// TIA Portal V20 export
FUNCTION "CollectAlarms" : Void   // FC62, LAD
TITLE = Alarm Collector Unit
// Collects alarms from the respective level and categorises the alarms into the different alarm classes.
// stored: Namespace Unit1, SetENOAutomatically false
   VAR_INPUT
      resetAlarms : Bool;
      disableAlarms : Bool;
   END_VAR
   VAR_OUTPUT
      commandsToUnit : "LUC_typeStateCommands";   // Feedback to the unit
   END_VAR
   VAR_TEMP
      interfaceUnuse : Array[0..1] of Bool;
      otherUnitError : Array[0..1] of Bool;
   END_VAR
   VAR CONSTANT
      TRUE : Bool := true;
      DelayTime : Time := T#300ms;
   END_VAR
BEGIN

REGION Network 1: Reset Alarms
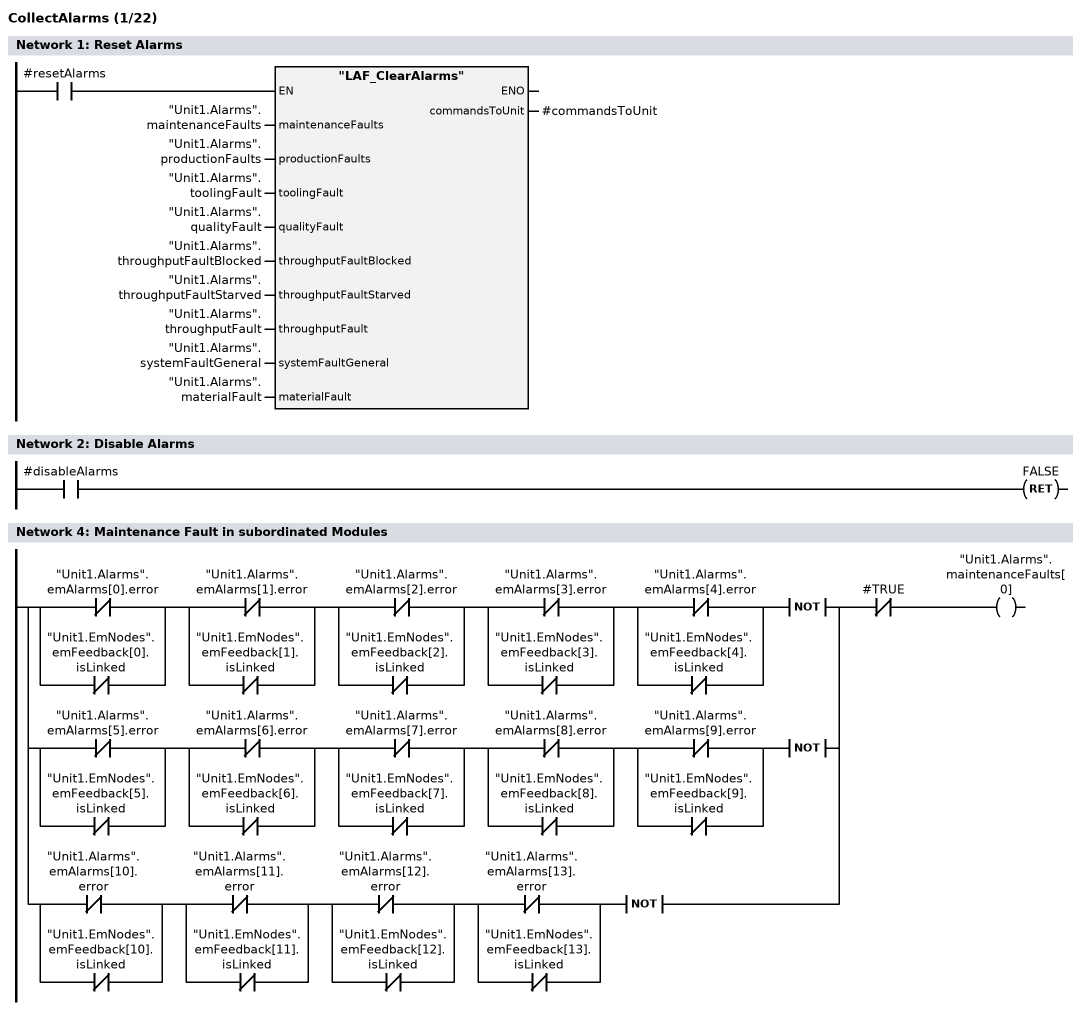
   RUNG wire#powerrail
      Contact( #resetAlarms )
      "LAF_ClearAlarms"(maintenanceFaults := "Unit1.Alarms".maintenanceFaults, productionFaults := "Unit1.Alarms".productionFaults, toolingFault := "Unit1.Alarms".toolingFault, qualityFault := "Unit1.Alarms".qualityFault, throughputFaultBlocked := "Unit1.Alarms".throughputFaultBlocked, throughputFaultStarved := "Unit1.Alarms".throughputFaultStarved, throughputFault := "Unit1.Alarms".throughputFault, systemFaultGeneral := "Unit1.Alarms".systemFaultGeneral, materialFault := "Unit1.Alarms".materialFault, commandsToUnit => #commandsToUnit)
   END_RUNG
   // the same network as SCL:
   IF #resetAlarms THEN
       "LAF_ClearAlarms"(maintenanceFaults := "Unit1.Alarms".maintenanceFaults,
                         productionFaults := "Unit1.Alarms".productionFaults,
                         toolingFault := "Unit1.Alarms".toolingFault,
                         qualityFault := "Unit1.Alarms".qualityFault,
                         throughputFaultBlocked := "Unit1.Alarms".throughputFaultBlocked,
                         throughputFaultStarved := "Unit1.Alarms".throughputFaultStarved,
                         throughputFault := "Unit1.Alarms".throughputFault,
                         systemFaultGeneral := "Unit1.Alarms".systemFaultGeneral,
                         materialFault := "Unit1.Alarms".materialFault,
                         commandsToUnit => #commandsToUnit);
   END_IF;
END_REGION

REGION Network 2: Disable Alarms
   RUNG wire#powerrail
      Contact( #disableAlarms )
      ReturnCoil( FALSE )
   END_RUNG
   // the same network as SCL:
   IF #disableAlarms THEN
       ENO := FALSE;
       RETURN;
   END_IF;
END_REGION

REGION Network 3: *************** Fault ************************
END_REGION

REGION Network 4: Maintenance Fault in subordinated Modules
   RUNG wire#powerrail
      I_Contact( "Unit1.Alarms".emAlarms[0].error )
      wire#w1
      I_Contact( "Unit1.Alarms".emAlarms[1].error )
      wire#w2
      I_Contact( "Unit1.Alarms".emAlarms[2].error )
      wire#w3
      I_Contact( "Unit1.Alarms".emAlarms[3].error )
      wire#w4
      I_Contact( "Unit1.Alarms".emAlarms[4].error )
      wire#w5
      Not()
      wire#w6
      I_Contact( #TRUE )
      Coil( "Unit1.Alarms".maintenanceFaults[0] )
   END_RUNG
   RUNG wire#powerrail
      I_Contact( "Unit1.EmNodes".emFeedback[0].isLinked )
   END_RUNG wire#w1
   RUNG wire#w1
      I_Contact( "Unit1.EmNodes".emFeedback[1].isLinked )
   END_RUNG wire#w2
   RUNG wire#w2
      I_Contact( "Unit1.EmNodes".emFeedback[2].isLinked )
   END_RUNG wire#w3
   RUNG wire#w3
      I_Contact( "Unit1.EmNodes".emFeedback[3].isLinked )
   END_RUNG wire#w4
   RUNG wire#w4
      I_Contact( "Unit1.EmNodes".emFeedback[4].isLinked )
   END_RUNG wire#w5
   RUNG wire#powerrail
      I_Contact( "Unit1.Alarms".emAlarms[5].error )
      wire#w7
      I_Contact( "Unit1.Alarms".emAlarms[6].error )
      wire#w8
      I_Contact( "Unit1.Alarms".emAlarms[7].error )
      wire#w9
      I_Contact( "Unit1.Alarms".emAlarms[8].error )
      wire#w10
      I_Contact( "Unit1.Alarms".emAlarms[9].error )
      wire#w11
      Not()
   END_RUNG wire#w6
   RUNG wire#powerrail
      I_Contact( "Unit1.EmNodes".emFeedback[5].isLinked )
   END_RUNG wire#w7
   RUNG wire#w7
      I_Contact( "Unit1.EmNodes".emFeedback[6].isLinked )
   END_RUNG wire#w8
   RUNG wire#w8
      I_Contact( "Unit1.EmNodes".emFeedback[7].isLinked )
   END_RUNG wire#w9
   RUNG wire#w9
      I_Contact( "Unit1.EmNodes".emFeedback[8].isLinked )
   END_RUNG wire#w10
   RUNG wire#w10
      I_Contact( "Unit1.EmNodes".emFeedback[9].isLinked )
   END_RUNG wire#w11
   RUNG wire#powerrail
      I_Contact( "Unit1.Alarms".emAlarms[10].error )
      wire#w12
      I_Contact( "Unit1.Alarms".emAlarms[11].error )
      wire#w13
      I_Contact( "Unit1.Alarms".emAlarms[12].error )
      wire#w14
      I_Contact( "Unit1.Alarms".emAlarms[13].error )
      wire#w15
      Not()
   END_RUNG wire#w6
   RUNG wire#powerrail
      I_Contact( "Unit1.EmNodes".emFeedback[10].isLinked )
   END_RUNG wire#w12
   RUNG wire#w12
      I_Contact( "Unit1.EmNodes".emFeedback[11].isLinked )
   END_RUNG wire#w13
   RUNG wire#w13
      I_Contact( "Unit1.EmNodes".emFeedback[12].isLinked )
   END_RUNG wire#w14
   RUNG wire#w14
      I_Contact( "Unit1.EmNodes".emFeedback[13].isLinked )
   END_RUNG wire#w15
   // the same network as SCL:
   "Unit1.Alarms".maintenanceFaults[0] := (NOT ((NOT "Unit1.Alarms".emAlarms[0].error OR NOT "Unit1.EmNodes".emFeedback[0].isLinked) AND (NOT "Unit1.Alarms".emAlarms[1].error OR NOT "Unit1.EmNodes".emFeedback[1].isLinked) AND (NOT "Unit1.Alarms".emAlarms[2].error OR NOT "Unit1.EmNodes".emFeedback[2].isLinked) AND (NOT "Unit1.Alarms".emAlarms[3].error OR NOT "Unit1.EmNodes".emFeedback[3].isLinked) AND (NOT "Unit1.Alarms".emAlarms[4].error OR NOT "Unit1.EmNodes".emFeedback[4].isLinked)) OR NOT ((NOT "Unit1.Alarms".emAlarms[5].error OR NOT "Unit1.EmNodes".emFeedback[5].isLinked) AND (NOT "Unit1.Alarms".emAlarms[6].error OR NOT "Unit1.EmNodes".emFeedback[6].isLinked) AND (NOT "Unit1.Alarms".emAlarms[7].error OR NOT "Unit1.EmNodes".emFeedback[7].isLinked) AND (NOT "Unit1.Alarms".emAlarms[8].error OR NOT "Unit1.EmNodes".emFeedback[8].isLinked) AND (NOT "Unit1.Alarms".emAlarms[9].error OR NOT "Unit1.EmNodes".emFeedback[9].isLinked)) OR NOT ((NOT "Unit1.Alarms".emAlarms[10].error OR NOT "Unit1.EmNodes".emFeedback[10].isLinked) AND (NOT "Unit1.Alarms".emAlarms[11].error OR NOT "Unit1.EmNodes".emFeedback[11].isLinked) AND (NOT "Unit1.Alarms".emAlarms[12].error OR NOT "Unit1.EmNodes".emFeedback[12].isLinked) AND (NOT "Unit1.Alarms".emAlarms[13].error OR NOT "Unit1.EmNodes".emFeedback[13].isLinked))) AND NOT #TRUE;
END_REGION

REGION Network 5: PFE Maintenance Faults 0 ~ 29
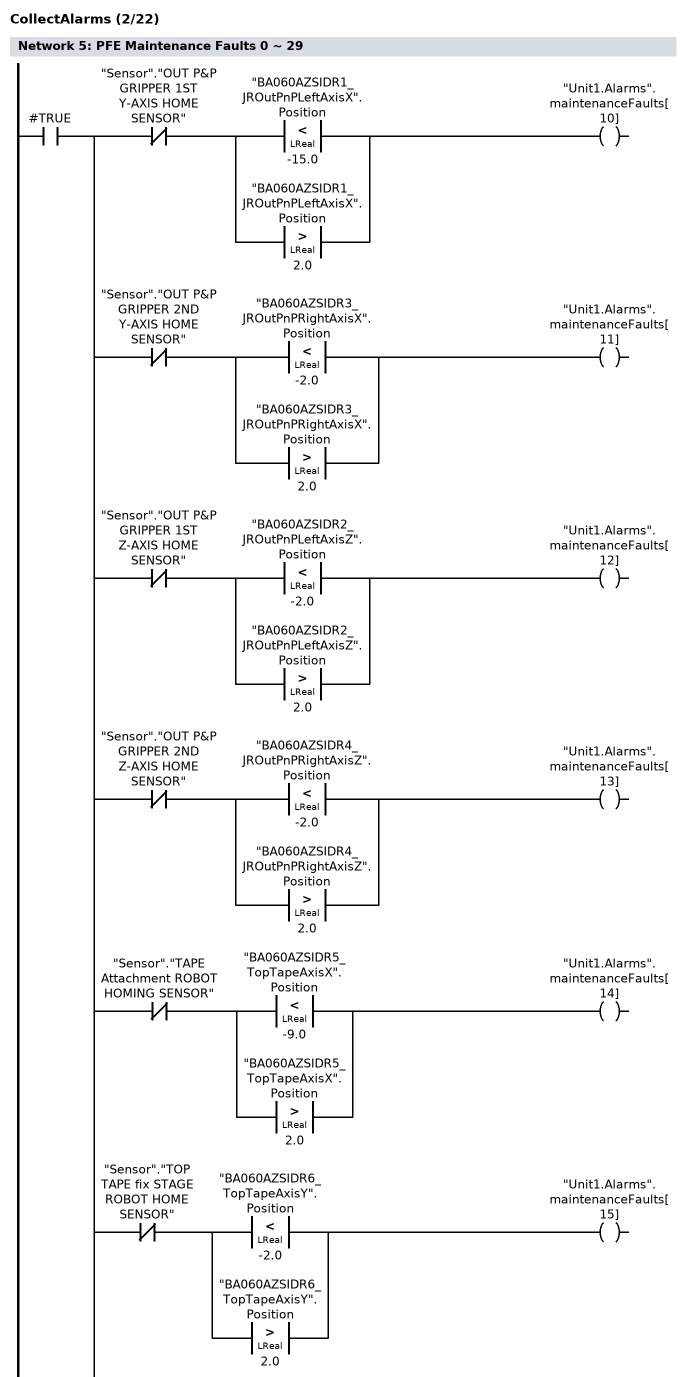
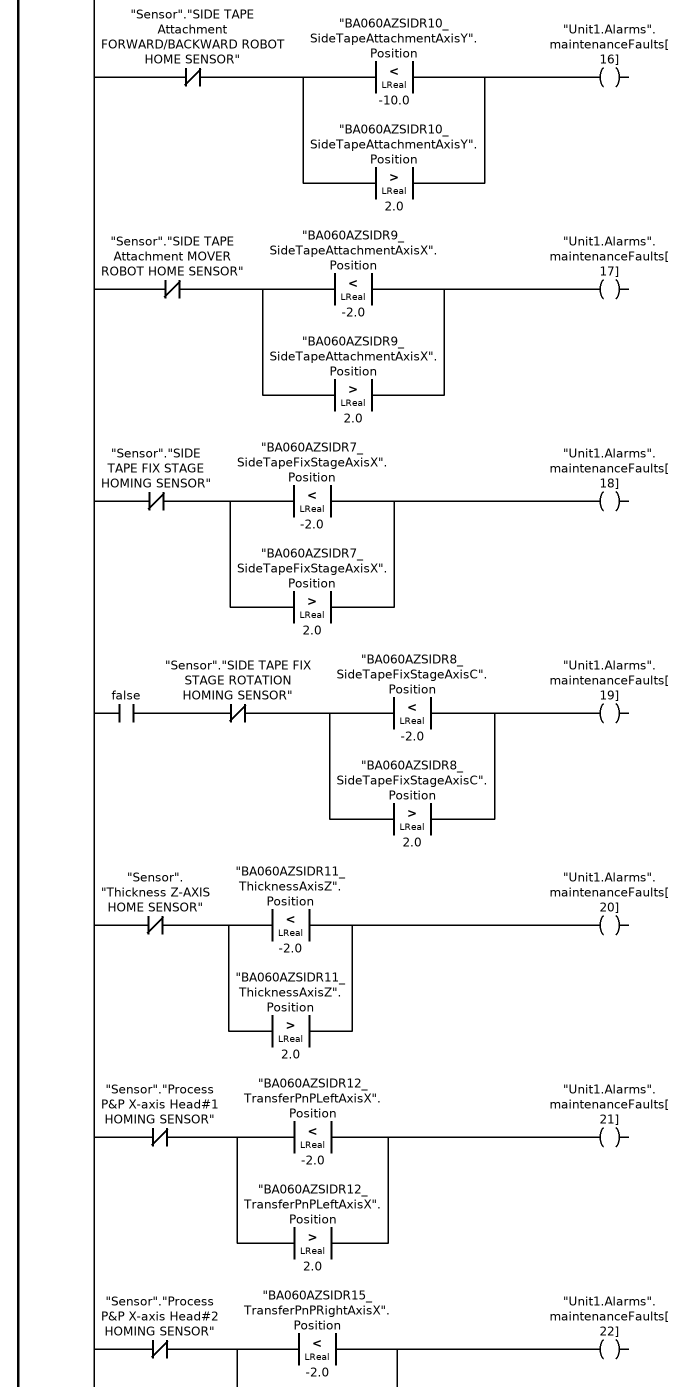
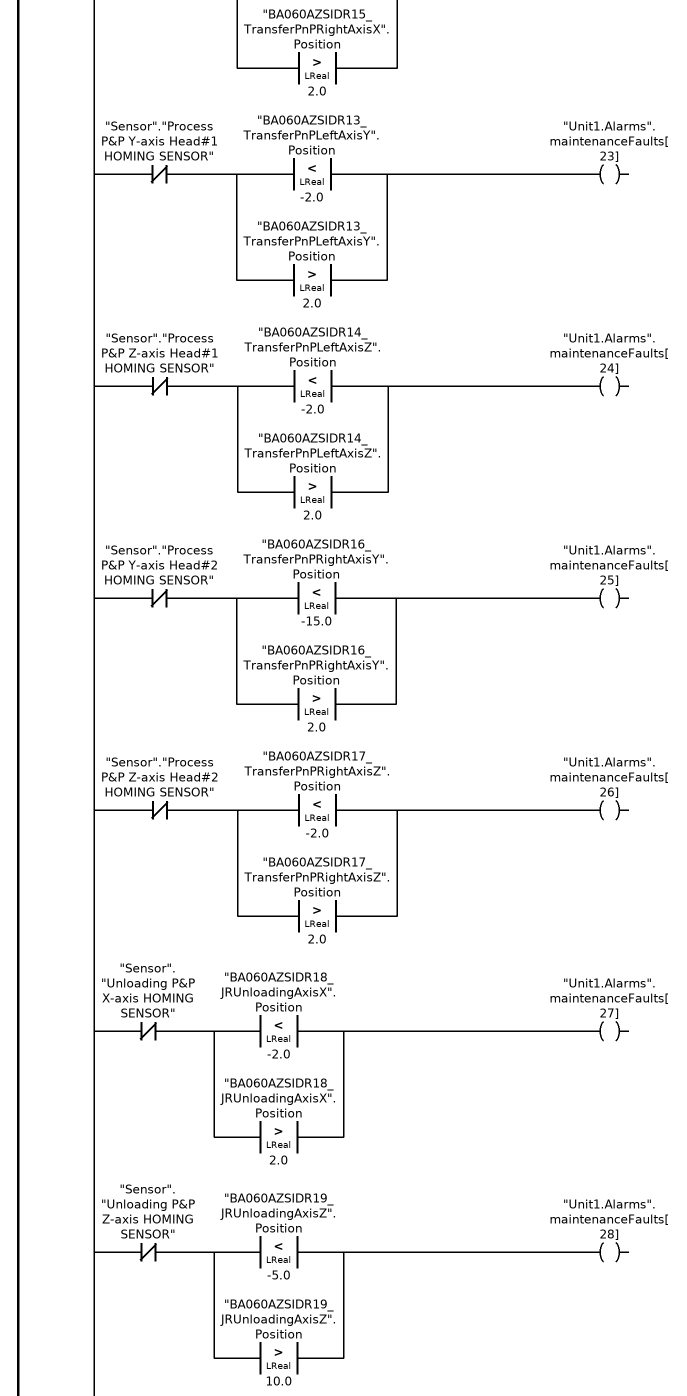
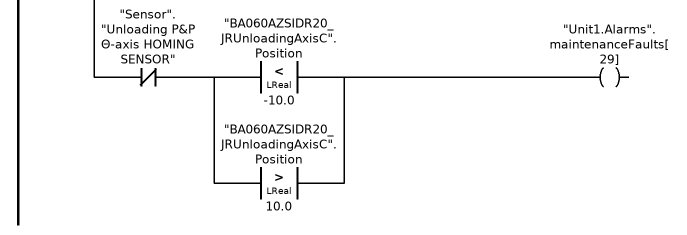
   RUNG wire#powerrail
      Contact( #TRUE )
      wire#w1
      I_Contact( "Sensor"."OUT P&P GRIPPER 1ST Y-AXIS HOME SENSOR" )
      wire#w2
      { S7_Templates := "SrcType := LReal" } LT_Contact(in1 := "BA060AZSIDR1_JROutPnPLeftAxisX".Position, in2 := -15.0)
      wire#w3
      Coil( "Unit1.Alarms".maintenanceFaults[10] )
   END_RUNG
   RUNG wire#w2
      { S7_Templates := "SrcType := LReal" } GT_Contact(in1 := "BA060AZSIDR1_JROutPnPLeftAxisX".Position, in2 := 2.0)
   END_RUNG wire#w3
   RUNG wire#w1
      I_Contact( "Sensor"."OUT P&P GRIPPER 2ND Y-AXIS HOME SENSOR" )
      wire#w4
      { S7_Templates := "SrcType := LReal" } LT_Contact(in1 := "BA060AZSIDR3_JROutPnPRightAxisX".Position, in2 := -2.0)
      wire#w5
      Coil( "Unit1.Alarms".maintenanceFaults[11] )
   END_RUNG
   RUNG wire#w4
      { S7_Templates := "SrcType := LReal" } GT_Contact(in1 := "BA060AZSIDR3_JROutPnPRightAxisX".Position, in2 := 2.0)
   END_RUNG wire#w5
   RUNG wire#w1
      I_Contact( "Sensor"."OUT P&P GRIPPER 1ST Z-AXIS HOME SENSOR" )
      wire#w6
      { S7_Templates := "SrcType := LReal" } LT_Contact(in1 := "BA060AZSIDR2_JROutPnPLeftAxisZ".Position, in2 := -2.0)
      wire#w7
      Coil( "Unit1.Alarms".maintenanceFaults[12] )
   END_RUNG
   RUNG wire#w6
      { S7_Templates := "SrcType := LReal" } GT_Contact(in1 := "BA060AZSIDR2_JROutPnPLeftAxisZ".Position, in2 := 2.0)
   END_RUNG wire#w7
   RUNG wire#w1
      I_Contact( "Sensor"."OUT P&P GRIPPER 2ND Z-AXIS HOME SENSOR" )
      wire#w8
      { S7_Templates := "SrcType := LReal" } LT_Contact(in1 := "BA060AZSIDR4_JROutPnPRightAxisZ".Position, in2 := -2.0)
      wire#w9
      Coil( "Unit1.Alarms".maintenanceFaults[13] )
   END_RUNG
   RUNG wire#w8
      { S7_Templates := "SrcType := LReal" } GT_Contact(in1 := "BA060AZSIDR4_JROutPnPRightAxisZ".Position, in2 := 2.0)
   END_RUNG wire#w9
   RUNG wire#w1
      I_Contact( "Sensor"."TAPE  Attachment ROBOT HOMING SENSOR" )
      wire#w10
      { S7_Templates := "SrcType := LReal" } LT_Contact(in1 := "BA060AZSIDR5_TopTapeAxisX".Position, in2 := -9.0)
      wire#w11
      Coil( "Unit1.Alarms".maintenanceFaults[14] )
   END_RUNG
   RUNG wire#w10
      { S7_Templates := "SrcType := LReal" } GT_Contact(in1 := "BA060AZSIDR5_TopTapeAxisX".Position, in2 := 2.0)
   END_RUNG wire#w11
   RUNG wire#w1
      I_Contact( "Sensor"."TOP TAPE fix STAGE ROBOT HOME SENSOR" )
      wire#w12
      { S7_Templates := "SrcType := LReal" } LT_Contact(in1 := "BA060AZSIDR6_TopTapeAxisY".Position, in2 := -2.0)
      wire#w13
      Coil( "Unit1.Alarms".maintenanceFaults[15] )
   END_RUNG
   RUNG wire#w12
      { S7_Templates := "SrcType := LReal" } GT_Contact(in1 := "BA060AZSIDR6_TopTapeAxisY".Position, in2 := 2.0)
   END_RUNG wire#w13
   RUNG wire#w1
      I_Contact( "Sensor"."SIDE TAPE Attachment FORWARD/BACKWARD ROBOT HOME SENSOR" )
      wire#w14
      { S7_Templates := "SrcType := LReal" } LT_Contact(in1 := "BA060AZSIDR10_SideTapeAttachmentAxisY".Position, in2 := -10.0)
      wire#w15
      Coil( "Unit1.Alarms".maintenanceFaults[16] )
   END_RUNG
   RUNG wire#w14
      { S7_Templates := "SrcType := LReal" } GT_Contact(in1 := "BA060AZSIDR10_SideTapeAttachmentAxisY".Position, in2 := 2.0)
   END_RUNG wire#w15
   RUNG wire#w1
      I_Contact( "Sensor"."SIDE TAPE Attachment MOVER ROBOT HOME SENSOR" )
      wire#w16
      { S7_Templates := "SrcType := LReal" } LT_Contact(in1 := "BA060AZSIDR9_SideTapeAttachmentAxisX".Position, in2 := -2.0)
      wire#w17
      Coil( "Unit1.Alarms".maintenanceFaults[17] )
   END_RUNG
   RUNG wire#w16
      { S7_Templates := "SrcType := LReal" } GT_Contact(in1 := "BA060AZSIDR9_SideTapeAttachmentAxisX".Position, in2 := 2.0)
   END_RUNG wire#w17
   RUNG wire#w1
      I_Contact( "Sensor"."SIDE TAPE FIX STAGE HOMING SENSOR" )
      wire#w18
      { S7_Templates := "SrcType := LReal" } LT_Contact(in1 := "BA060AZSIDR7_SideTapeFixStageAxisX".Position, in2 := -2.0)
      wire#w19
      Coil( "Unit1.Alarms".maintenanceFaults[18] )
   END_RUNG
   RUNG wire#w18
      { S7_Templates := "SrcType := LReal" } GT_Contact(in1 := "BA060AZSIDR7_SideTapeFixStageAxisX".Position, in2 := 2.0)
   END_RUNG wire#w19
   RUNG wire#w1
      Contact( false )
      I_Contact( "Sensor"."SIDE TAPE FIX STAGE ROTATION HOMING SENSOR" )
      wire#w20
      { S7_Templates := "SrcType := LReal" } LT_Contact(in1 := "BA060AZSIDR8_SideTapeFixStageAxisC".Position, in2 := -2.0)
      wire#w21
      Coil( "Unit1.Alarms".maintenanceFaults[19] )
   END_RUNG
   RUNG wire#w20
      { S7_Templates := "SrcType := LReal" } GT_Contact(in1 := "BA060AZSIDR8_SideTapeFixStageAxisC".Position, in2 := 2.0)
   END_RUNG wire#w21
   RUNG wire#w1
      I_Contact( "Sensor"."Thickness Z-AXIS HOME SENSOR" )
      wire#w22
      { S7_Templates := "SrcType := LReal" } LT_Contact(in1 := "BA060AZSIDR11_ThicknessAxisZ".Position, in2 := -2.0)
      wire#w23
      Coil( "Unit1.Alarms".maintenanceFaults[20] )
   END_RUNG
   RUNG wire#w22
      { S7_Templates := "SrcType := LReal" } GT_Contact(in1 := "BA060AZSIDR11_ThicknessAxisZ".Position, in2 := 2.0)
   END_RUNG wire#w23
   RUNG wire#w1
      I_Contact( "Sensor"."Process P&P X-axis Head#1 HOMING SENSOR" )
      wire#w24
      { S7_Templates := "SrcType := LReal" } LT_Contact(in1 := "BA060AZSIDR12_TransferPnPLeftAxisX".Position, in2 := -2.0)
      wire#w25
      Coil( "Unit1.Alarms".maintenanceFaults[21] )
   END_RUNG
   RUNG wire#w24
      { S7_Templates := "SrcType := LReal" } GT_Contact(in1 := "BA060AZSIDR12_TransferPnPLeftAxisX".Position, in2 := 2.0)
   END_RUNG wire#w25
   RUNG wire#w1
      I_Contact( "Sensor"."Process P&P X-axis Head#2 HOMING SENSOR" )
      wire#w26
      { S7_Templates := "SrcType := LReal" } LT_Contact(in1 := "BA060AZSIDR15_TransferPnPRightAxisX".Position, in2 := -2.0)
      wire#w27
      Coil( "Unit1.Alarms".maintenanceFaults[22] )
   END_RUNG
   RUNG wire#w26
      { S7_Templates := "SrcType := LReal" } GT_Contact(in1 := "BA060AZSIDR15_TransferPnPRightAxisX".Position, in2 := 2.0)
   END_RUNG wire#w27
   RUNG wire#w1
      I_Contact( "Sensor"."Process P&P Y-axis Head#1 HOMING SENSOR" )
      wire#w28
      { S7_Templates := "SrcType := LReal" } LT_Contact(in1 := "BA060AZSIDR13_TransferPnPLeftAxisY".Position, in2 := -2.0)
      wire#w29
      Coil( "Unit1.Alarms".maintenanceFaults[23] )
   END_RUNG
   RUNG wire#w28
      { S7_Templates := "SrcType := LReal" } GT_Contact(in1 := "BA060AZSIDR13_TransferPnPLeftAxisY".Position, in2 := 2.0)
   END_RUNG wire#w29
   RUNG wire#w1
      I_Contact( "Sensor"."Process P&P Z-axis Head#1 HOMING SENSOR" )
      wire#w30
      { S7_Templates := "SrcType := LReal" } LT_Contact(in1 := "BA060AZSIDR14_TransferPnPLeftAxisZ".Position, in2 := -2.0)
      wire#w31
      Coil( "Unit1.Alarms".maintenanceFaults[24] )
   END_RUNG
   RUNG wire#w30
      { S7_Templates := "SrcType := LReal" } GT_Contact(in1 := "BA060AZSIDR14_TransferPnPLeftAxisZ".Position, in2 := 2.0)
   END_RUNG wire#w31
   RUNG wire#w1
      I_Contact( "Sensor"."Process P&P Y-axis Head#2 HOMING SENSOR" )
      wire#w32
      { S7_Templates := "SrcType := LReal" } LT_Contact(in1 := "BA060AZSIDR16_TransferPnPRightAxisY".Position, in2 := -15.0)
      wire#w33
      Coil( "Unit1.Alarms".maintenanceFaults[25] )
   END_RUNG
   RUNG wire#w32
      { S7_Templates := "SrcType := LReal" } GT_Contact(in1 := "BA060AZSIDR16_TransferPnPRightAxisY".Position, in2 := 2.0)
   END_RUNG wire#w33
   RUNG wire#w1
      I_Contact( "Sensor"."Process P&P Z-axis Head#2 HOMING SENSOR" )
      wire#w34
      { S7_Templates := "SrcType := LReal" } LT_Contact(in1 := "BA060AZSIDR17_TransferPnPRightAxisZ".Position, in2 := -2.0)
      wire#w35
      Coil( "Unit1.Alarms".maintenanceFaults[26] )
   END_RUNG
   RUNG wire#w34
      { S7_Templates := "SrcType := LReal" } GT_Contact(in1 := "BA060AZSIDR17_TransferPnPRightAxisZ".Position, in2 := 2.0)
   END_RUNG wire#w35
   RUNG wire#w1
      I_Contact( "Sensor"."Unloading P&P X-axis HOMING SENSOR" )
      wire#w36
      { S7_Templates := "SrcType := LReal" } LT_Contact(in1 := "BA060AZSIDR18_JRUnloadingAxisX".Position, in2 := -2.0)
      wire#w37
      Coil( "Unit1.Alarms".maintenanceFaults[27] )
   END_RUNG
   RUNG wire#w36
      { S7_Templates := "SrcType := LReal" } GT_Contact(in1 := "BA060AZSIDR18_JRUnloadingAxisX".Position, in2 := 2.0)
   END_RUNG wire#w37
   RUNG wire#w1
      I_Contact( "Sensor"."Unloading P&P Z-axis HOMING SENSOR" )
      wire#w38
      { S7_Templates := "SrcType := LReal" } LT_Contact(in1 := "BA060AZSIDR19_JRUnloadingAxisZ".Position, in2 := -5.0)
      wire#w39
      Coil( "Unit1.Alarms".maintenanceFaults[28] )
   END_RUNG
   RUNG wire#w38
      { S7_Templates := "SrcType := LReal" } GT_Contact(in1 := "BA060AZSIDR19_JRUnloadingAxisZ".Position, in2 := 10.0)
   END_RUNG wire#w39
   RUNG wire#w1
      I_Contact( "Sensor"."Unloading P&P Θ-axis HOMING SENSOR" )
      wire#w40
      { S7_Templates := "SrcType := LReal" } LT_Contact(in1 := "BA060AZSIDR20_JRUnloadingAxisC".Position, in2 := -10.0)
      wire#w41
      Coil( "Unit1.Alarms".maintenanceFaults[29] )
   END_RUNG
   RUNG wire#w40
      { S7_Templates := "SrcType := LReal" } GT_Contact(in1 := "BA060AZSIDR20_JRUnloadingAxisC".Position, in2 := 10.0)
   END_RUNG wire#w41
   // the same network as SCL:
   "Unit1.Alarms".maintenanceFaults[10] := #TRUE AND NOT "Sensor"."OUT P&P GRIPPER 1ST Y-AXIS HOME SENSOR" AND (("BA060AZSIDR1_JROutPnPLeftAxisX".Position < (-15.0)) OR ("BA060AZSIDR1_JROutPnPLeftAxisX".Position > 2.0));
   "Unit1.Alarms".maintenanceFaults[11] := #TRUE AND NOT "Sensor"."OUT P&P GRIPPER 2ND Y-AXIS HOME SENSOR" AND (("BA060AZSIDR3_JROutPnPRightAxisX".Position < (-2.0)) OR ("BA060AZSIDR3_JROutPnPRightAxisX".Position > 2.0));
   "Unit1.Alarms".maintenanceFaults[12] := #TRUE AND NOT "Sensor"."OUT P&P GRIPPER 1ST Z-AXIS HOME SENSOR" AND (("BA060AZSIDR2_JROutPnPLeftAxisZ".Position < (-2.0)) OR ("BA060AZSIDR2_JROutPnPLeftAxisZ".Position > 2.0));
   "Unit1.Alarms".maintenanceFaults[13] := #TRUE AND NOT "Sensor"."OUT P&P GRIPPER 2ND Z-AXIS HOME SENSOR" AND (("BA060AZSIDR4_JROutPnPRightAxisZ".Position < (-2.0)) OR ("BA060AZSIDR4_JROutPnPRightAxisZ".Position > 2.0));
   "Unit1.Alarms".maintenanceFaults[14] := #TRUE AND NOT "Sensor"."TAPE  Attachment ROBOT HOMING SENSOR" AND (("BA060AZSIDR5_TopTapeAxisX".Position < (-9.0)) OR ("BA060AZSIDR5_TopTapeAxisX".Position > 2.0));
   "Unit1.Alarms".maintenanceFaults[15] := #TRUE AND NOT "Sensor"."TOP TAPE fix STAGE ROBOT HOME SENSOR" AND (("BA060AZSIDR6_TopTapeAxisY".Position < (-2.0)) OR ("BA060AZSIDR6_TopTapeAxisY".Position > 2.0));
   "Unit1.Alarms".maintenanceFaults[16] := #TRUE AND NOT "Sensor"."SIDE TAPE Attachment FORWARD/BACKWARD ROBOT HOME SENSOR" AND (("BA060AZSIDR10_SideTapeAttachmentAxisY".Position < (-10.0)) OR ("BA060AZSIDR10_SideTapeAttachmentAxisY".Position > 2.0));
   "Unit1.Alarms".maintenanceFaults[17] := #TRUE AND NOT "Sensor"."SIDE TAPE Attachment MOVER ROBOT HOME SENSOR" AND (("BA060AZSIDR9_SideTapeAttachmentAxisX".Position < (-2.0)) OR ("BA060AZSIDR9_SideTapeAttachmentAxisX".Position > 2.0));
   "Unit1.Alarms".maintenanceFaults[18] := #TRUE AND NOT "Sensor"."SIDE TAPE FIX STAGE HOMING SENSOR" AND (("BA060AZSIDR7_SideTapeFixStageAxisX".Position < (-2.0)) OR ("BA060AZSIDR7_SideTapeFixStageAxisX".Position > 2.0));
   "Unit1.Alarms".maintenanceFaults[19] := #TRUE AND false AND NOT "Sensor"."SIDE TAPE FIX STAGE ROTATION HOMING SENSOR" AND (("BA060AZSIDR8_SideTapeFixStageAxisC".Position < (-2.0)) OR ("BA060AZSIDR8_SideTapeFixStageAxisC".Position > 2.0));
   "Unit1.Alarms".maintenanceFaults[20] := #TRUE AND NOT "Sensor"."Thickness Z-AXIS HOME SENSOR" AND (("BA060AZSIDR11_ThicknessAxisZ".Position < (-2.0)) OR ("BA060AZSIDR11_ThicknessAxisZ".Position > 2.0));
   "Unit1.Alarms".maintenanceFaults[21] := #TRUE AND NOT "Sensor"."Process P&P X-axis Head#1 HOMING SENSOR" AND (("BA060AZSIDR12_TransferPnPLeftAxisX".Position < (-2.0)) OR ("BA060AZSIDR12_TransferPnPLeftAxisX".Position > 2.0));
   "Unit1.Alarms".maintenanceFaults[22] := #TRUE AND NOT "Sensor"."Process P&P X-axis Head#2 HOMING SENSOR" AND (("BA060AZSIDR15_TransferPnPRightAxisX".Position < (-2.0)) OR ("BA060AZSIDR15_TransferPnPRightAxisX".Position > 2.0));
   "Unit1.Alarms".maintenanceFaults[23] := #TRUE AND NOT "Sensor"."Process P&P Y-axis Head#1 HOMING SENSOR" AND (("BA060AZSIDR13_TransferPnPLeftAxisY".Position < (-2.0)) OR ("BA060AZSIDR13_TransferPnPLeftAxisY".Position > 2.0));
   "Unit1.Alarms".maintenanceFaults[24] := #TRUE AND NOT "Sensor"."Process P&P Z-axis Head#1 HOMING SENSOR" AND (("BA060AZSIDR14_TransferPnPLeftAxisZ".Position < (-2.0)) OR ("BA060AZSIDR14_TransferPnPLeftAxisZ".Position > 2.0));
   "Unit1.Alarms".maintenanceFaults[25] := #TRUE AND NOT "Sensor"."Process P&P Y-axis Head#2 HOMING SENSOR" AND (("BA060AZSIDR16_TransferPnPRightAxisY".Position < (-15.0)) OR ("BA060AZSIDR16_TransferPnPRightAxisY".Position > 2.0));
   "Unit1.Alarms".maintenanceFaults[26] := #TRUE AND NOT "Sensor"."Process P&P Z-axis Head#2 HOMING SENSOR" AND (("BA060AZSIDR17_TransferPnPRightAxisZ".Position < (-2.0)) OR ("BA060AZSIDR17_TransferPnPRightAxisZ".Position > 2.0));
   "Unit1.Alarms".maintenanceFaults[27] := #TRUE AND NOT "Sensor"."Unloading P&P X-axis HOMING SENSOR" AND (("BA060AZSIDR18_JRUnloadingAxisX".Position < (-2.0)) OR ("BA060AZSIDR18_JRUnloadingAxisX".Position > 2.0));
   "Unit1.Alarms".maintenanceFaults[28] := #TRUE AND NOT "Sensor"."Unloading P&P Z-axis HOMING SENSOR" AND (("BA060AZSIDR19_JRUnloadingAxisZ".Position < (-5.0)) OR ("BA060AZSIDR19_JRUnloadingAxisZ".Position > 10.0));
   "Unit1.Alarms".maintenanceFaults[29] := #TRUE AND NOT "Sensor"."Unloading P&P Θ-axis HOMING SENSOR" AND (("BA060AZSIDR20_JRUnloadingAxisC".Position < (-10.0)) OR ("BA060AZSIDR20_JRUnloadingAxisC".Position > 10.0));
END_REGION

REGION Network 6: PFE Maintenance Faults 30
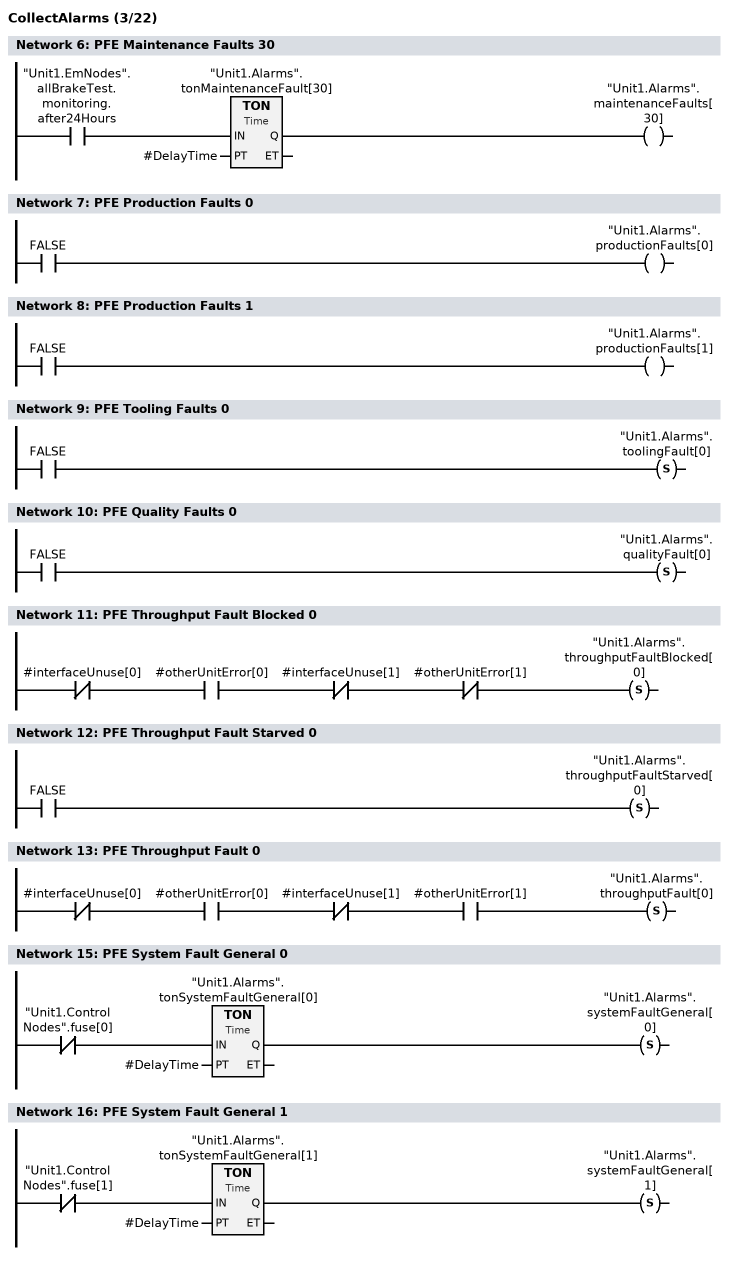
   RUNG wire#powerrail
      Contact( "Unit1.EmNodes".allBrakeTest.monitoring.after24Hours )
      { S7_Templates := "time_type := Time" } "Unit1.Alarms".tonMaintenanceFault[30].TON(pt := #DelayTime, et =>)
      Coil( "Unit1.Alarms".maintenanceFaults[30] )
   END_RUNG
   // the same network as SCL:
   "Unit1.Alarms".tonMaintenanceFault[30].TON(IN := "Unit1.EmNodes".allBrakeTest.monitoring.after24Hours,
                           PT := #DelayTime);
   "Unit1.Alarms".maintenanceFaults[30] := "Unit1.Alarms".tonMaintenanceFault[30].Q;
END_REGION

REGION Network 7: PFE Production Faults 0
   RUNG wire#powerrail
      Contact( FALSE )
      Coil( "Unit1.Alarms".productionFaults[0] )
   END_RUNG
   // the same network as SCL:
   "Unit1.Alarms".productionFaults[0] := FALSE;
END_REGION

REGION Network 8: PFE Production Faults 1
   RUNG wire#powerrail
      Contact( FALSE )
      Coil( "Unit1.Alarms".productionFaults[1] )
   END_RUNG
   // the same network as SCL:
   "Unit1.Alarms".productionFaults[1] := FALSE;
END_REGION

REGION Network 9: PFE Tooling Faults 0
   RUNG wire#powerrail
      Contact( FALSE )
      S_Coil( "Unit1.Alarms".toolingFault[0] )
   END_RUNG
   // the same network as SCL:
   IF FALSE THEN "Unit1.Alarms".toolingFault[0] := TRUE; END_IF;
END_REGION

REGION Network 10: PFE Quality Faults 0
   RUNG wire#powerrail
      Contact( FALSE )
      S_Coil( "Unit1.Alarms".qualityFault[0] )
   END_RUNG
   // the same network as SCL:
   IF FALSE THEN "Unit1.Alarms".qualityFault[0] := TRUE; END_IF;
END_REGION

REGION Network 11: PFE Throughput Fault Blocked 0
   RUNG wire#powerrail
      I_Contact( #interfaceUnuse[0] )
      Contact( #otherUnitError[0] )
      I_Contact( #interfaceUnuse[1] )
      I_Contact( #otherUnitError[1] )
      S_Coil( "Unit1.Alarms".throughputFaultBlocked[0] )
   END_RUNG
   // the same network as SCL:
   IF NOT #interfaceUnuse[0] AND #otherUnitError[0] AND NOT #interfaceUnuse[1] AND NOT #otherUnitError[1] THEN
       "Unit1.Alarms".throughputFaultBlocked[0] := TRUE;
   END_IF;
END_REGION

REGION Network 12: PFE Throughput Fault Starved 0
   RUNG wire#powerrail
      Contact( FALSE )
      S_Coil( "Unit1.Alarms".throughputFaultStarved[0] )
   END_RUNG
   // the same network as SCL:
   IF FALSE THEN "Unit1.Alarms".throughputFaultStarved[0] := TRUE; END_IF;
END_REGION

REGION Network 13: PFE Throughput Fault 0
   RUNG wire#powerrail
      I_Contact( #interfaceUnuse[0] )
      Contact( #otherUnitError[0] )
      I_Contact( #interfaceUnuse[1] )
      Contact( #otherUnitError[1] )
      S_Coil( "Unit1.Alarms".throughputFault[0] )
   END_RUNG
   // the same network as SCL:
   IF NOT #interfaceUnuse[0] AND #otherUnitError[0] AND NOT #interfaceUnuse[1] AND #otherUnitError[1] THEN
       "Unit1.Alarms".throughputFault[0] := TRUE;
   END_IF;
END_REGION

REGION Network 14 (SCL): PFE System Fault General Spare
   //Alarms.systemFaultGeneral[3] := NOT ControlNodes.fusess[3]; //SPARE
   //Alarms.systemFaultGeneral[4] := NOT ControlNodes.fusess[4]; //SPARE
   //Alarms.systemFaultGeneral[10] := NOT ControlNodes.fusess[10]; //SPARE
   //Alarms.systemFaultGeneral[12] := NOT ControlNodes.fusess[12]; //SPARE
   //Alarms.systemFaultGeneral[18] := NOT ControlNodes.fusess[18]; //SPARE
   //Alarms.systemFaultGeneral[19] := NOT ControlNodes.fusess[19]; //SPARE
   //Alarms.systemFaultGeneral[25] := NOT ControlNodes.fusess[25]; //SPRE
   //Alarms.systemFaultGeneral[27] := NOT ControlNodes.fusess[27]; //SPARE
   //Alarms.systemFaultGeneral[28] := NOT ControlNodes.fusess[28]; //SPARE
   //Alarms.systemFaultGeneral[34] := NOT ControlNodes.fusess[34]; //SPARE
   //Alarms.systemFaultGeneral[54] := NOT ControlNodes.fusess[54]; //SPARE
   //Alarms.systemFaultGeneral[63] := NOT ControlNodes.fusess[63]; //SPARE
   //Alarms.systemFaultGeneral[73] := NOT ControlNodes.fusess[73]; //SPARE
   //Alarms.systemFaultGeneral[79] := NOT ControlNodes.fusess[79]; //SPARE
   //Alarms.systemFaultGeneral[84] := NOT ControlNodes.fuse[84]; //SPARE
   //Alarms.systemFaultGeneral[118] := NOT ControlNodes.fusess[118]; //SPARE
   //Alarms.systemFaultGeneral[119] := NOT ControlNodes.fusess[119]; //SPARE
   //Alarms.systemFaultGeneral[120] := NOT ControlNodes.fusess[120]; //SPARE
   //Alarms.systemFaultGeneral[121] := NOT ControlNodes.fusess[121]; //SPARE
END_REGION

REGION Network 15: PFE System Fault General 0
   RUNG wire#powerrail
      I_Contact( "Unit1.ControlNodes".fuse[0] )
      { S7_Templates := "time_type := Time" } "Unit1.Alarms".tonSystemFaultGeneral[0].TON(pt := #DelayTime, et =>)
      S_Coil( "Unit1.Alarms".systemFaultGeneral[0] )
   END_RUNG
   // the same network as SCL:
   "Unit1.Alarms".tonSystemFaultGeneral[0].TON(IN := NOT "Unit1.ControlNodes".fuse[0], PT := #DelayTime);
   IF "Unit1.Alarms".tonSystemFaultGeneral[0].Q THEN "Unit1.Alarms".systemFaultGeneral[0] := TRUE; END_IF;
END_REGION

REGION Network 16: PFE System Fault General 1
   RUNG wire#powerrail
      I_Contact( "Unit1.ControlNodes".fuse[1] )
      { S7_Templates := "time_type := Time" } "Unit1.Alarms".tonSystemFaultGeneral[1].TON(pt := #DelayTime, et =>)
      S_Coil( "Unit1.Alarms".systemFaultGeneral[1] )
   END_RUNG
   // the same network as SCL:
   "Unit1.Alarms".tonSystemFaultGeneral[1].TON(IN := NOT "Unit1.ControlNodes".fuse[1], PT := #DelayTime);
   IF "Unit1.Alarms".tonSystemFaultGeneral[1].Q THEN "Unit1.Alarms".systemFaultGeneral[1] := TRUE; END_IF;
END_REGION

REGION Network 17: PFE System Fault General 2
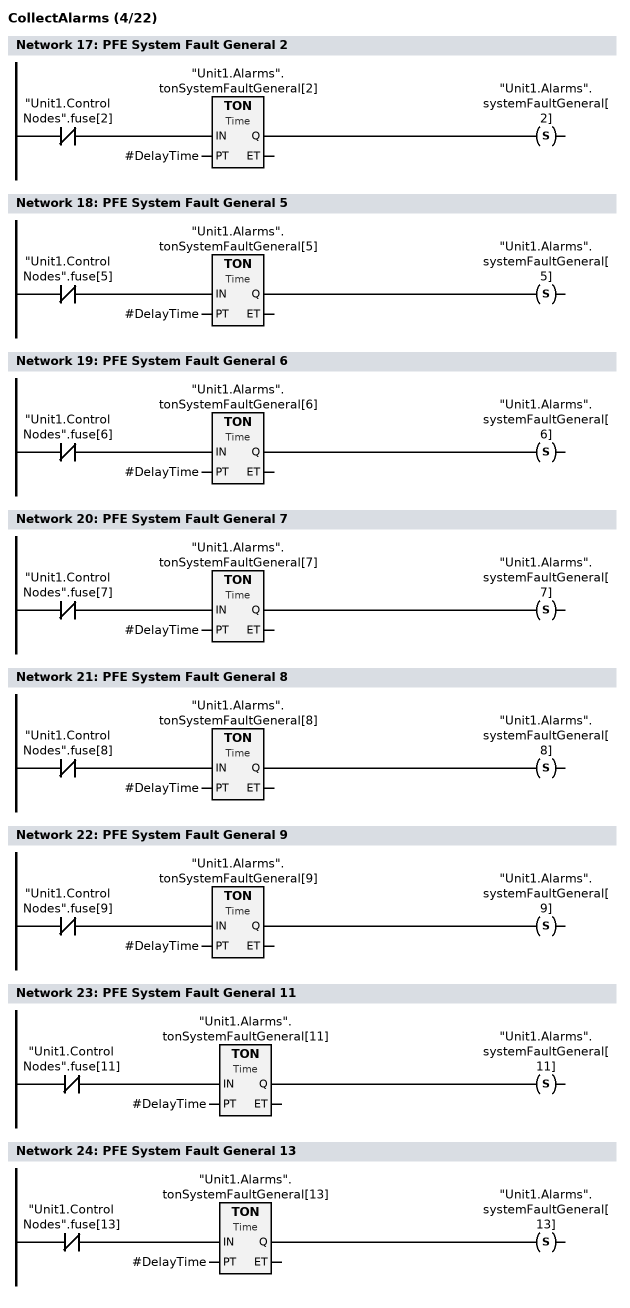
   RUNG wire#powerrail
      I_Contact( "Unit1.ControlNodes".fuse[2] )
      { S7_Templates := "time_type := Time" } "Unit1.Alarms".tonSystemFaultGeneral[2].TON(pt := #DelayTime, et =>)
      S_Coil( "Unit1.Alarms".systemFaultGeneral[2] )
   END_RUNG
   // the same network as SCL:
   "Unit1.Alarms".tonSystemFaultGeneral[2].TON(IN := NOT "Unit1.ControlNodes".fuse[2], PT := #DelayTime);
   IF "Unit1.Alarms".tonSystemFaultGeneral[2].Q THEN "Unit1.Alarms".systemFaultGeneral[2] := TRUE; END_IF;
END_REGION

REGION Network 18: PFE System Fault General 5
   RUNG wire#powerrail
      I_Contact( "Unit1.ControlNodes".fuse[5] )
      { S7_Templates := "time_type := Time" } "Unit1.Alarms".tonSystemFaultGeneral[5].TON(pt := #DelayTime, et =>)
      S_Coil( "Unit1.Alarms".systemFaultGeneral[5] )
   END_RUNG
   // the same network as SCL:
   "Unit1.Alarms".tonSystemFaultGeneral[5].TON(IN := NOT "Unit1.ControlNodes".fuse[5], PT := #DelayTime);
   IF "Unit1.Alarms".tonSystemFaultGeneral[5].Q THEN "Unit1.Alarms".systemFaultGeneral[5] := TRUE; END_IF;
END_REGION

REGION Network 19: PFE System Fault General 6
   RUNG wire#powerrail
      I_Contact( "Unit1.ControlNodes".fuse[6] )
      { S7_Templates := "time_type := Time" } "Unit1.Alarms".tonSystemFaultGeneral[6].TON(pt := #DelayTime, et =>)
      S_Coil( "Unit1.Alarms".systemFaultGeneral[6] )
   END_RUNG
   // the same network as SCL:
   "Unit1.Alarms".tonSystemFaultGeneral[6].TON(IN := NOT "Unit1.ControlNodes".fuse[6], PT := #DelayTime);
   IF "Unit1.Alarms".tonSystemFaultGeneral[6].Q THEN "Unit1.Alarms".systemFaultGeneral[6] := TRUE; END_IF;
END_REGION

REGION Network 20: PFE System Fault General 7
   RUNG wire#powerrail
      I_Contact( "Unit1.ControlNodes".fuse[7] )
      { S7_Templates := "time_type := Time" } "Unit1.Alarms".tonSystemFaultGeneral[7].TON(pt := #DelayTime, et =>)
      S_Coil( "Unit1.Alarms".systemFaultGeneral[7] )
   END_RUNG
   // the same network as SCL:
   "Unit1.Alarms".tonSystemFaultGeneral[7].TON(IN := NOT "Unit1.ControlNodes".fuse[7], PT := #DelayTime);
   IF "Unit1.Alarms".tonSystemFaultGeneral[7].Q THEN "Unit1.Alarms".systemFaultGeneral[7] := TRUE; END_IF;
END_REGION

REGION Network 21: PFE System Fault General 8
   RUNG wire#powerrail
      I_Contact( "Unit1.ControlNodes".fuse[8] )
      { S7_Templates := "time_type := Time" } "Unit1.Alarms".tonSystemFaultGeneral[8].TON(pt := #DelayTime, et =>)
      S_Coil( "Unit1.Alarms".systemFaultGeneral[8] )
   END_RUNG
   // the same network as SCL:
   "Unit1.Alarms".tonSystemFaultGeneral[8].TON(IN := NOT "Unit1.ControlNodes".fuse[8], PT := #DelayTime);
   IF "Unit1.Alarms".tonSystemFaultGeneral[8].Q THEN "Unit1.Alarms".systemFaultGeneral[8] := TRUE; END_IF;
END_REGION

REGION Network 22: PFE System Fault General 9
   RUNG wire#powerrail
      I_Contact( "Unit1.ControlNodes".fuse[9] )
      { S7_Templates := "time_type := Time" } "Unit1.Alarms".tonSystemFaultGeneral[9].TON(pt := #DelayTime, et =>)
      S_Coil( "Unit1.Alarms".systemFaultGeneral[9] )
   END_RUNG
   // the same network as SCL:
   "Unit1.Alarms".tonSystemFaultGeneral[9].TON(IN := NOT "Unit1.ControlNodes".fuse[9], PT := #DelayTime);
   IF "Unit1.Alarms".tonSystemFaultGeneral[9].Q THEN "Unit1.Alarms".systemFaultGeneral[9] := TRUE; END_IF;
END_REGION

REGION Network 23: PFE System Fault General 11
   RUNG wire#powerrail
      I_Contact( "Unit1.ControlNodes".fuse[11] )
      { S7_Templates := "time_type := Time" } "Unit1.Alarms".tonSystemFaultGeneral[11].TON(pt := #DelayTime, et =>)
      S_Coil( "Unit1.Alarms".systemFaultGeneral[11] )
   END_RUNG
   // the same network as SCL:
   "Unit1.Alarms".tonSystemFaultGeneral[11].TON(IN := NOT "Unit1.ControlNodes".fuse[11], PT := #DelayTime);
   IF "Unit1.Alarms".tonSystemFaultGeneral[11].Q THEN "Unit1.Alarms".systemFaultGeneral[11] := TRUE; END_IF;
END_REGION

REGION Network 24: PFE System Fault General 13
   RUNG wire#powerrail
      I_Contact( "Unit1.ControlNodes".fuse[13] )
      { S7_Templates := "time_type := Time" } "Unit1.Alarms".tonSystemFaultGeneral[13].TON(pt := #DelayTime, et =>)
      S_Coil( "Unit1.Alarms".systemFaultGeneral[13] )
   END_RUNG
   // the same network as SCL:
   "Unit1.Alarms".tonSystemFaultGeneral[13].TON(IN := NOT "Unit1.ControlNodes".fuse[13], PT := #DelayTime);
   IF "Unit1.Alarms".tonSystemFaultGeneral[13].Q THEN "Unit1.Alarms".systemFaultGeneral[13] := TRUE; END_IF;
END_REGION

REGION Network 25: PFE System Fault General 14
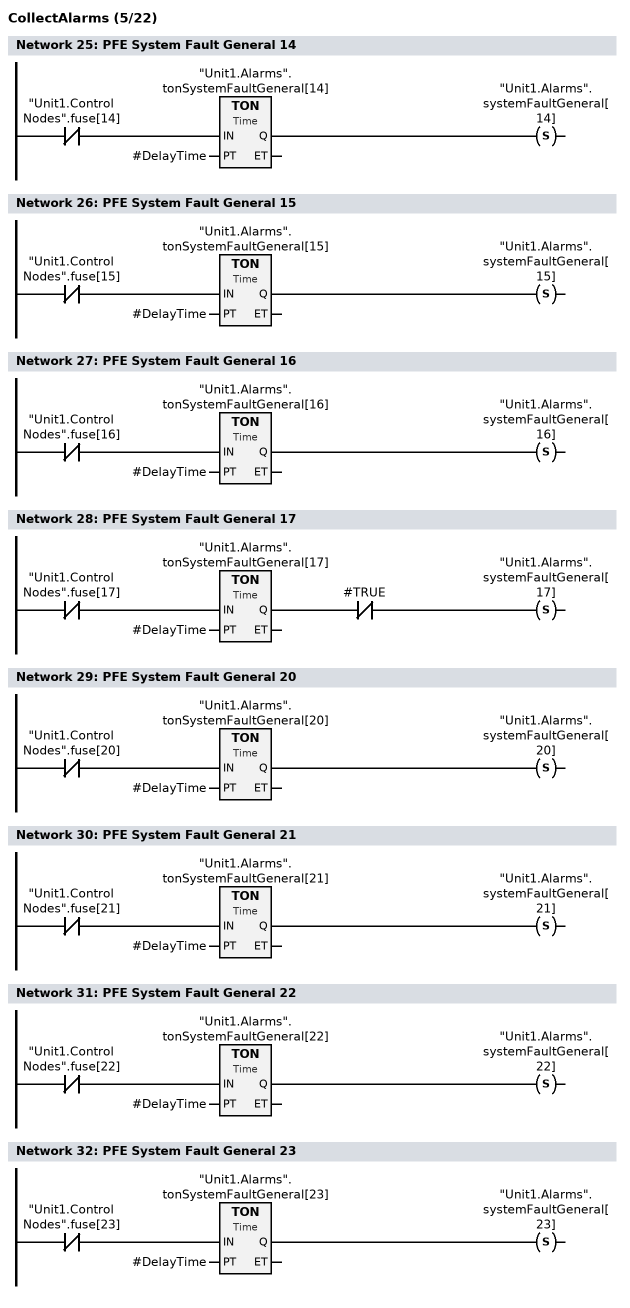
   RUNG wire#powerrail
      I_Contact( "Unit1.ControlNodes".fuse[14] )
      { S7_Templates := "time_type := Time" } "Unit1.Alarms".tonSystemFaultGeneral[14].TON(pt := #DelayTime, et =>)
      S_Coil( "Unit1.Alarms".systemFaultGeneral[14] )
   END_RUNG
   // the same network as SCL:
   "Unit1.Alarms".tonSystemFaultGeneral[14].TON(IN := NOT "Unit1.ControlNodes".fuse[14], PT := #DelayTime);
   IF "Unit1.Alarms".tonSystemFaultGeneral[14].Q THEN "Unit1.Alarms".systemFaultGeneral[14] := TRUE; END_IF;
END_REGION

REGION Network 26: PFE System Fault General 15
   RUNG wire#powerrail
      I_Contact( "Unit1.ControlNodes".fuse[15] )
      { S7_Templates := "time_type := Time" } "Unit1.Alarms".tonSystemFaultGeneral[15].TON(pt := #DelayTime, et =>)
      S_Coil( "Unit1.Alarms".systemFaultGeneral[15] )
   END_RUNG
   // the same network as SCL:
   "Unit1.Alarms".tonSystemFaultGeneral[15].TON(IN := NOT "Unit1.ControlNodes".fuse[15], PT := #DelayTime);
   IF "Unit1.Alarms".tonSystemFaultGeneral[15].Q THEN "Unit1.Alarms".systemFaultGeneral[15] := TRUE; END_IF;
END_REGION

REGION Network 27: PFE System Fault General 16
   RUNG wire#powerrail
      I_Contact( "Unit1.ControlNodes".fuse[16] )
      { S7_Templates := "time_type := Time" } "Unit1.Alarms".tonSystemFaultGeneral[16].TON(pt := #DelayTime, et =>)
      S_Coil( "Unit1.Alarms".systemFaultGeneral[16] )
   END_RUNG
   // the same network as SCL:
   "Unit1.Alarms".tonSystemFaultGeneral[16].TON(IN := NOT "Unit1.ControlNodes".fuse[16], PT := #DelayTime);
   IF "Unit1.Alarms".tonSystemFaultGeneral[16].Q THEN "Unit1.Alarms".systemFaultGeneral[16] := TRUE; END_IF;
END_REGION

REGION Network 28: PFE System Fault General 17
   RUNG wire#powerrail
      I_Contact( "Unit1.ControlNodes".fuse[17] )
      { S7_Templates := "time_type := Time" } "Unit1.Alarms".tonSystemFaultGeneral[17].TON(pt := #DelayTime, et =>)
      I_Contact( #TRUE )
      S_Coil( "Unit1.Alarms".systemFaultGeneral[17] )
   END_RUNG
   // the same network as SCL:
   "Unit1.Alarms".tonSystemFaultGeneral[17].TON(IN := NOT "Unit1.ControlNodes".fuse[17], PT := #DelayTime);
   IF "Unit1.Alarms".tonSystemFaultGeneral[17].Q AND NOT #TRUE THEN
       "Unit1.Alarms".systemFaultGeneral[17] := TRUE;
   END_IF;
END_REGION

REGION Network 29: PFE System Fault General 20
   RUNG wire#powerrail
      I_Contact( "Unit1.ControlNodes".fuse[20] )
      { S7_Templates := "time_type := Time" } "Unit1.Alarms".tonSystemFaultGeneral[20].TON(pt := #DelayTime, et =>)
      S_Coil( "Unit1.Alarms".systemFaultGeneral[20] )
   END_RUNG
   // the same network as SCL:
   "Unit1.Alarms".tonSystemFaultGeneral[20].TON(IN := NOT "Unit1.ControlNodes".fuse[20], PT := #DelayTime);
   IF "Unit1.Alarms".tonSystemFaultGeneral[20].Q THEN "Unit1.Alarms".systemFaultGeneral[20] := TRUE; END_IF;
END_REGION

REGION Network 30: PFE System Fault General 21
   RUNG wire#powerrail
      I_Contact( "Unit1.ControlNodes".fuse[21] )
      { S7_Templates := "time_type := Time" } "Unit1.Alarms".tonSystemFaultGeneral[21].TON(pt := #DelayTime, et =>)
      S_Coil( "Unit1.Alarms".systemFaultGeneral[21] )
   END_RUNG
   // the same network as SCL:
   "Unit1.Alarms".tonSystemFaultGeneral[21].TON(IN := NOT "Unit1.ControlNodes".fuse[21], PT := #DelayTime);
   IF "Unit1.Alarms".tonSystemFaultGeneral[21].Q THEN "Unit1.Alarms".systemFaultGeneral[21] := TRUE; END_IF;
END_REGION

REGION Network 31: PFE System Fault General 22
   RUNG wire#powerrail
      I_Contact( "Unit1.ControlNodes".fuse[22] )
      { S7_Templates := "time_type := Time" } "Unit1.Alarms".tonSystemFaultGeneral[22].TON(pt := #DelayTime, et =>)
      S_Coil( "Unit1.Alarms".systemFaultGeneral[22] )
   END_RUNG
   // the same network as SCL:
   "Unit1.Alarms".tonSystemFaultGeneral[22].TON(IN := NOT "Unit1.ControlNodes".fuse[22], PT := #DelayTime);
   IF "Unit1.Alarms".tonSystemFaultGeneral[22].Q THEN "Unit1.Alarms".systemFaultGeneral[22] := TRUE; END_IF;
END_REGION

REGION Network 32: PFE System Fault General 23
   RUNG wire#powerrail
      I_Contact( "Unit1.ControlNodes".fuse[23] )
      { S7_Templates := "time_type := Time" } "Unit1.Alarms".tonSystemFaultGeneral[23].TON(pt := #DelayTime, et =>)
      S_Coil( "Unit1.Alarms".systemFaultGeneral[23] )
   END_RUNG
   // the same network as SCL:
   "Unit1.Alarms".tonSystemFaultGeneral[23].TON(IN := NOT "Unit1.ControlNodes".fuse[23], PT := #DelayTime);
   IF "Unit1.Alarms".tonSystemFaultGeneral[23].Q THEN "Unit1.Alarms".systemFaultGeneral[23] := TRUE; END_IF;
END_REGION

REGION Network 33: PFE System Fault General 24
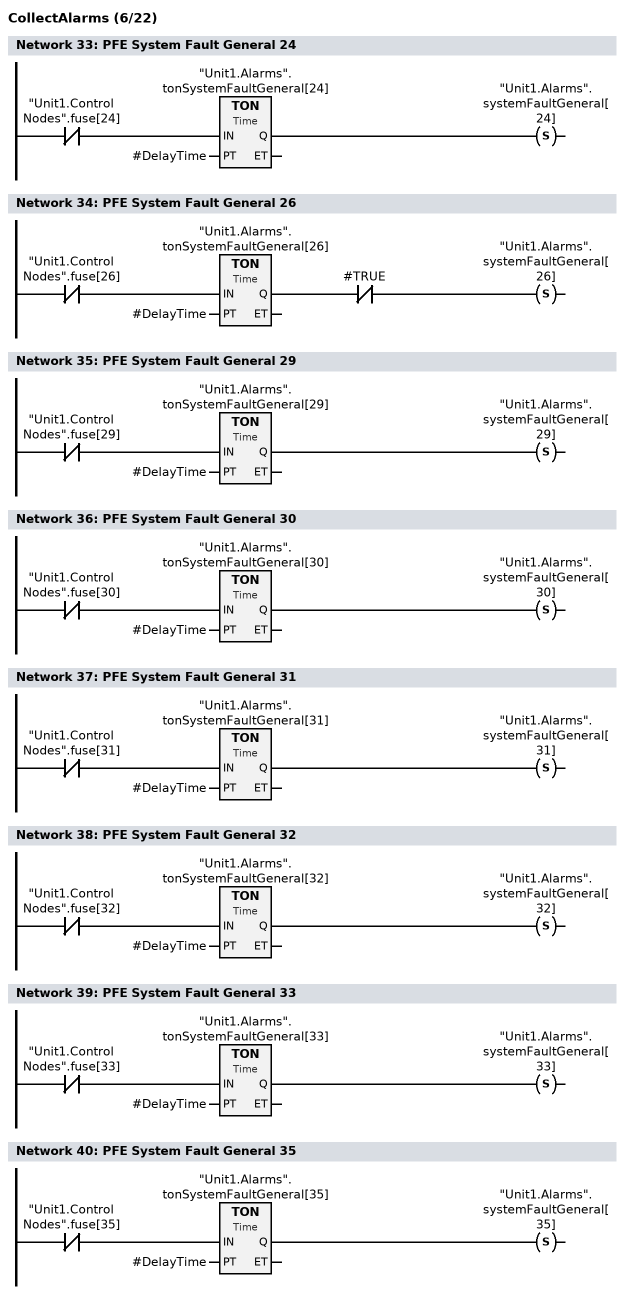
   RUNG wire#powerrail
      I_Contact( "Unit1.ControlNodes".fuse[24] )
      { S7_Templates := "time_type := Time" } "Unit1.Alarms".tonSystemFaultGeneral[24].TON(pt := #DelayTime, et =>)
      S_Coil( "Unit1.Alarms".systemFaultGeneral[24] )
   END_RUNG
   // the same network as SCL:
   "Unit1.Alarms".tonSystemFaultGeneral[24].TON(IN := NOT "Unit1.ControlNodes".fuse[24], PT := #DelayTime);
   IF "Unit1.Alarms".tonSystemFaultGeneral[24].Q THEN "Unit1.Alarms".systemFaultGeneral[24] := TRUE; END_IF;
END_REGION

REGION Network 34: PFE System Fault General 26
   RUNG wire#powerrail
      I_Contact( "Unit1.ControlNodes".fuse[26] )
      { S7_Templates := "time_type := Time" } "Unit1.Alarms".tonSystemFaultGeneral[26].TON(pt := #DelayTime, et =>)
      I_Contact( #TRUE )
      S_Coil( "Unit1.Alarms".systemFaultGeneral[26] )
   END_RUNG
   // the same network as SCL:
   "Unit1.Alarms".tonSystemFaultGeneral[26].TON(IN := NOT "Unit1.ControlNodes".fuse[26], PT := #DelayTime);
   IF "Unit1.Alarms".tonSystemFaultGeneral[26].Q AND NOT #TRUE THEN
       "Unit1.Alarms".systemFaultGeneral[26] := TRUE;
   END_IF;
END_REGION

REGION Network 35: PFE System Fault General 29
   RUNG wire#powerrail
      I_Contact( "Unit1.ControlNodes".fuse[29] )
      { S7_Templates := "time_type := Time" } "Unit1.Alarms".tonSystemFaultGeneral[29].TON(pt := #DelayTime, et =>)
      S_Coil( "Unit1.Alarms".systemFaultGeneral[29] )
   END_RUNG
   // the same network as SCL:
   "Unit1.Alarms".tonSystemFaultGeneral[29].TON(IN := NOT "Unit1.ControlNodes".fuse[29], PT := #DelayTime);
   IF "Unit1.Alarms".tonSystemFaultGeneral[29].Q THEN "Unit1.Alarms".systemFaultGeneral[29] := TRUE; END_IF;
END_REGION

REGION Network 36: PFE System Fault General 30
   RUNG wire#powerrail
      I_Contact( "Unit1.ControlNodes".fuse[30] )
      { S7_Templates := "time_type := Time" } "Unit1.Alarms".tonSystemFaultGeneral[30].TON(pt := #DelayTime, et =>)
      S_Coil( "Unit1.Alarms".systemFaultGeneral[30] )
   END_RUNG
   // the same network as SCL:
   "Unit1.Alarms".tonSystemFaultGeneral[30].TON(IN := NOT "Unit1.ControlNodes".fuse[30], PT := #DelayTime);
   IF "Unit1.Alarms".tonSystemFaultGeneral[30].Q THEN "Unit1.Alarms".systemFaultGeneral[30] := TRUE; END_IF;
END_REGION

REGION Network 37: PFE System Fault General 31
   RUNG wire#powerrail
      I_Contact( "Unit1.ControlNodes".fuse[31] )
      { S7_Templates := "time_type := Time" } "Unit1.Alarms".tonSystemFaultGeneral[31].TON(pt := #DelayTime, et =>)
      S_Coil( "Unit1.Alarms".systemFaultGeneral[31] )
   END_RUNG
   // the same network as SCL:
   "Unit1.Alarms".tonSystemFaultGeneral[31].TON(IN := NOT "Unit1.ControlNodes".fuse[31], PT := #DelayTime);
   IF "Unit1.Alarms".tonSystemFaultGeneral[31].Q THEN "Unit1.Alarms".systemFaultGeneral[31] := TRUE; END_IF;
END_REGION

REGION Network 38: PFE System Fault General 32
   RUNG wire#powerrail
      I_Contact( "Unit1.ControlNodes".fuse[32] )
      { S7_Templates := "time_type := Time" } "Unit1.Alarms".tonSystemFaultGeneral[32].TON(pt := #DelayTime, et =>)
      S_Coil( "Unit1.Alarms".systemFaultGeneral[32] )
   END_RUNG
   // the same network as SCL:
   "Unit1.Alarms".tonSystemFaultGeneral[32].TON(IN := NOT "Unit1.ControlNodes".fuse[32], PT := #DelayTime);
   IF "Unit1.Alarms".tonSystemFaultGeneral[32].Q THEN "Unit1.Alarms".systemFaultGeneral[32] := TRUE; END_IF;
END_REGION

REGION Network 39: PFE System Fault General 33
   RUNG wire#powerrail
      I_Contact( "Unit1.ControlNodes".fuse[33] )
      { S7_Templates := "time_type := Time" } "Unit1.Alarms".tonSystemFaultGeneral[33].TON(pt := #DelayTime, et =>)
      S_Coil( "Unit1.Alarms".systemFaultGeneral[33] )
   END_RUNG
   // the same network as SCL:
   "Unit1.Alarms".tonSystemFaultGeneral[33].TON(IN := NOT "Unit1.ControlNodes".fuse[33], PT := #DelayTime);
   IF "Unit1.Alarms".tonSystemFaultGeneral[33].Q THEN "Unit1.Alarms".systemFaultGeneral[33] := TRUE; END_IF;
END_REGION

REGION Network 40: PFE System Fault General 35
   RUNG wire#powerrail
      I_Contact( "Unit1.ControlNodes".fuse[35] )
      { S7_Templates := "time_type := Time" } "Unit1.Alarms".tonSystemFaultGeneral[35].TON(pt := #DelayTime, et =>)
      S_Coil( "Unit1.Alarms".systemFaultGeneral[35] )
   END_RUNG
   // the same network as SCL:
   "Unit1.Alarms".tonSystemFaultGeneral[35].TON(IN := NOT "Unit1.ControlNodes".fuse[35], PT := #DelayTime);
   IF "Unit1.Alarms".tonSystemFaultGeneral[35].Q THEN "Unit1.Alarms".systemFaultGeneral[35] := TRUE; END_IF;
END_REGION

REGION Network 41: PFE System Fault General 36
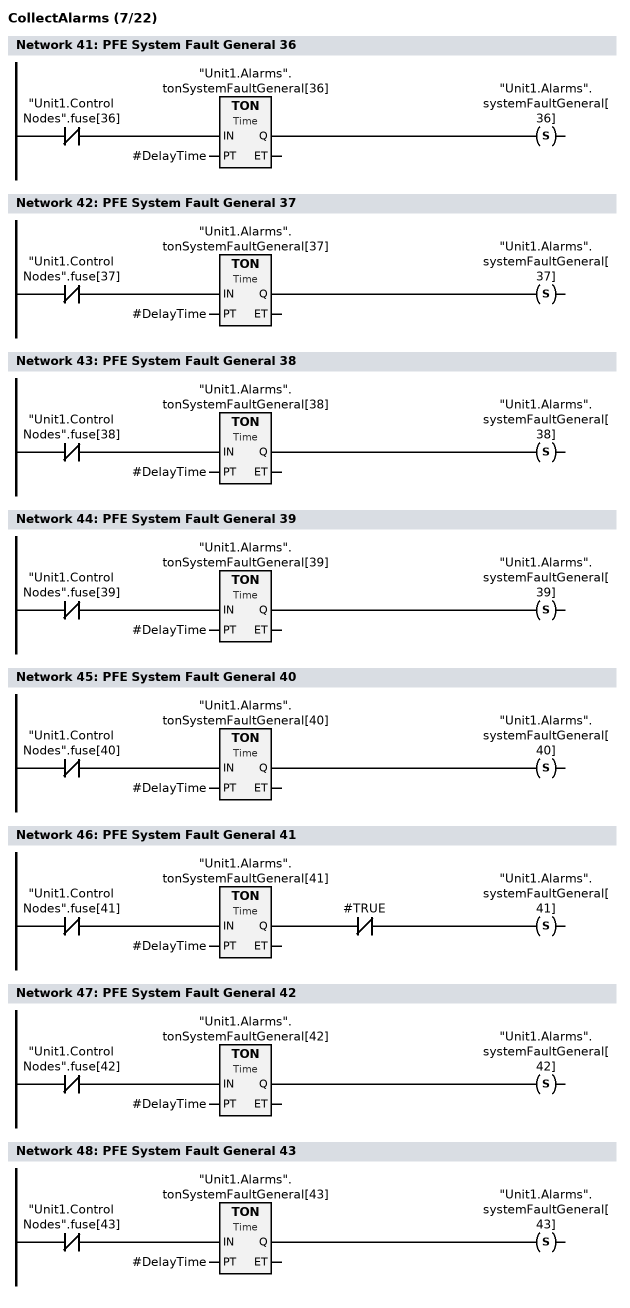
   RUNG wire#powerrail
      I_Contact( "Unit1.ControlNodes".fuse[36] )
      { S7_Templates := "time_type := Time" } "Unit1.Alarms".tonSystemFaultGeneral[36].TON(pt := #DelayTime, et =>)
      S_Coil( "Unit1.Alarms".systemFaultGeneral[36] )
   END_RUNG
   // the same network as SCL:
   "Unit1.Alarms".tonSystemFaultGeneral[36].TON(IN := NOT "Unit1.ControlNodes".fuse[36], PT := #DelayTime);
   IF "Unit1.Alarms".tonSystemFaultGeneral[36].Q THEN "Unit1.Alarms".systemFaultGeneral[36] := TRUE; END_IF;
END_REGION

REGION Network 42: PFE System Fault General 37
   RUNG wire#powerrail
      I_Contact( "Unit1.ControlNodes".fuse[37] )
      { S7_Templates := "time_type := Time" } "Unit1.Alarms".tonSystemFaultGeneral[37].TON(pt := #DelayTime, et =>)
      S_Coil( "Unit1.Alarms".systemFaultGeneral[37] )
   END_RUNG
   // the same network as SCL:
   "Unit1.Alarms".tonSystemFaultGeneral[37].TON(IN := NOT "Unit1.ControlNodes".fuse[37], PT := #DelayTime);
   IF "Unit1.Alarms".tonSystemFaultGeneral[37].Q THEN "Unit1.Alarms".systemFaultGeneral[37] := TRUE; END_IF;
END_REGION

REGION Network 43: PFE System Fault General 38
   RUNG wire#powerrail
      I_Contact( "Unit1.ControlNodes".fuse[38] )
      { S7_Templates := "time_type := Time" } "Unit1.Alarms".tonSystemFaultGeneral[38].TON(pt := #DelayTime, et =>)
      S_Coil( "Unit1.Alarms".systemFaultGeneral[38] )
   END_RUNG
   // the same network as SCL:
   "Unit1.Alarms".tonSystemFaultGeneral[38].TON(IN := NOT "Unit1.ControlNodes".fuse[38], PT := #DelayTime);
   IF "Unit1.Alarms".tonSystemFaultGeneral[38].Q THEN "Unit1.Alarms".systemFaultGeneral[38] := TRUE; END_IF;
END_REGION

REGION Network 44: PFE System Fault General 39
   RUNG wire#powerrail
      I_Contact( "Unit1.ControlNodes".fuse[39] )
      { S7_Templates := "time_type := Time" } "Unit1.Alarms".tonSystemFaultGeneral[39].TON(pt := #DelayTime, et =>)
      S_Coil( "Unit1.Alarms".systemFaultGeneral[39] )
   END_RUNG
   // the same network as SCL:
   "Unit1.Alarms".tonSystemFaultGeneral[39].TON(IN := NOT "Unit1.ControlNodes".fuse[39], PT := #DelayTime);
   IF "Unit1.Alarms".tonSystemFaultGeneral[39].Q THEN "Unit1.Alarms".systemFaultGeneral[39] := TRUE; END_IF;
END_REGION

REGION Network 45: PFE System Fault General 40
   RUNG wire#powerrail
      I_Contact( "Unit1.ControlNodes".fuse[40] )
      { S7_Templates := "time_type := Time" } "Unit1.Alarms".tonSystemFaultGeneral[40].TON(pt := #DelayTime, et =>)
      S_Coil( "Unit1.Alarms".systemFaultGeneral[40] )
   END_RUNG
   // the same network as SCL:
   "Unit1.Alarms".tonSystemFaultGeneral[40].TON(IN := NOT "Unit1.ControlNodes".fuse[40], PT := #DelayTime);
   IF "Unit1.Alarms".tonSystemFaultGeneral[40].Q THEN "Unit1.Alarms".systemFaultGeneral[40] := TRUE; END_IF;
END_REGION

REGION Network 46: PFE System Fault General 41
   RUNG wire#powerrail
      I_Contact( "Unit1.ControlNodes".fuse[41] )
      { S7_Templates := "time_type := Time" } "Unit1.Alarms".tonSystemFaultGeneral[41].TON(pt := #DelayTime, et =>)
      I_Contact( #TRUE )
      S_Coil( "Unit1.Alarms".systemFaultGeneral[41] )
   END_RUNG
   // the same network as SCL:
   "Unit1.Alarms".tonSystemFaultGeneral[41].TON(IN := NOT "Unit1.ControlNodes".fuse[41], PT := #DelayTime);
   IF "Unit1.Alarms".tonSystemFaultGeneral[41].Q AND NOT #TRUE THEN
       "Unit1.Alarms".systemFaultGeneral[41] := TRUE;
   END_IF;
END_REGION

REGION Network 47: PFE System Fault General 42
   RUNG wire#powerrail
      I_Contact( "Unit1.ControlNodes".fuse[42] )
      { S7_Templates := "time_type := Time" } "Unit1.Alarms".tonSystemFaultGeneral[42].TON(pt := #DelayTime, et =>)
      S_Coil( "Unit1.Alarms".systemFaultGeneral[42] )
   END_RUNG
   // the same network as SCL:
   "Unit1.Alarms".tonSystemFaultGeneral[42].TON(IN := NOT "Unit1.ControlNodes".fuse[42], PT := #DelayTime);
   IF "Unit1.Alarms".tonSystemFaultGeneral[42].Q THEN "Unit1.Alarms".systemFaultGeneral[42] := TRUE; END_IF;
END_REGION

REGION Network 48: PFE System Fault General 43
   RUNG wire#powerrail
      I_Contact( "Unit1.ControlNodes".fuse[43] )
      { S7_Templates := "time_type := Time" } "Unit1.Alarms".tonSystemFaultGeneral[43].TON(pt := #DelayTime, et =>)
      S_Coil( "Unit1.Alarms".systemFaultGeneral[43] )
   END_RUNG
   // the same network as SCL:
   "Unit1.Alarms".tonSystemFaultGeneral[43].TON(IN := NOT "Unit1.ControlNodes".fuse[43], PT := #DelayTime);
   IF "Unit1.Alarms".tonSystemFaultGeneral[43].Q THEN "Unit1.Alarms".systemFaultGeneral[43] := TRUE; END_IF;
END_REGION

REGION Network 49: PFE System Fault General 44
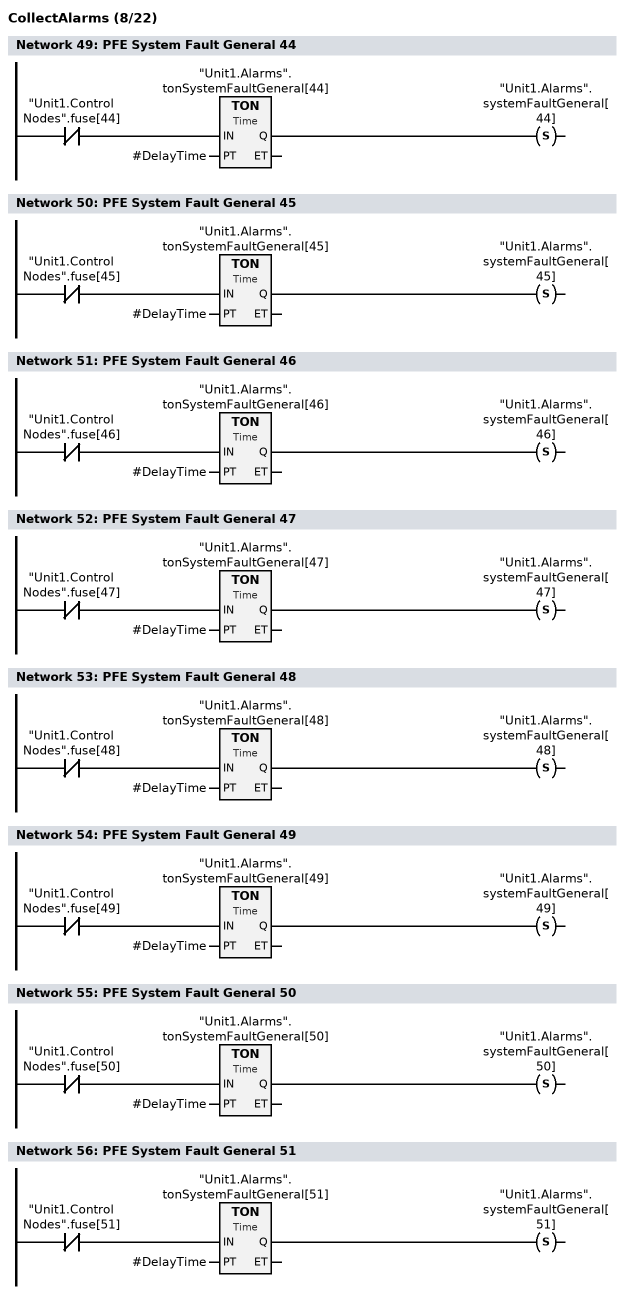
   RUNG wire#powerrail
      I_Contact( "Unit1.ControlNodes".fuse[44] )
      { S7_Templates := "time_type := Time" } "Unit1.Alarms".tonSystemFaultGeneral[44].TON(pt := #DelayTime, et =>)
      S_Coil( "Unit1.Alarms".systemFaultGeneral[44] )
   END_RUNG
   // the same network as SCL:
   "Unit1.Alarms".tonSystemFaultGeneral[44].TON(IN := NOT "Unit1.ControlNodes".fuse[44], PT := #DelayTime);
   IF "Unit1.Alarms".tonSystemFaultGeneral[44].Q THEN "Unit1.Alarms".systemFaultGeneral[44] := TRUE; END_IF;
END_REGION

REGION Network 50: PFE System Fault General 45
   RUNG wire#powerrail
      I_Contact( "Unit1.ControlNodes".fuse[45] )
      { S7_Templates := "time_type := Time" } "Unit1.Alarms".tonSystemFaultGeneral[45].TON(pt := #DelayTime, et =>)
      S_Coil( "Unit1.Alarms".systemFaultGeneral[45] )
   END_RUNG
   // the same network as SCL:
   "Unit1.Alarms".tonSystemFaultGeneral[45].TON(IN := NOT "Unit1.ControlNodes".fuse[45], PT := #DelayTime);
   IF "Unit1.Alarms".tonSystemFaultGeneral[45].Q THEN "Unit1.Alarms".systemFaultGeneral[45] := TRUE; END_IF;
END_REGION

REGION Network 51: PFE System Fault General 46
   RUNG wire#powerrail
      I_Contact( "Unit1.ControlNodes".fuse[46] )
      { S7_Templates := "time_type := Time" } "Unit1.Alarms".tonSystemFaultGeneral[46].TON(pt := #DelayTime, et =>)
      S_Coil( "Unit1.Alarms".systemFaultGeneral[46] )
   END_RUNG
   // the same network as SCL:
   "Unit1.Alarms".tonSystemFaultGeneral[46].TON(IN := NOT "Unit1.ControlNodes".fuse[46], PT := #DelayTime);
   IF "Unit1.Alarms".tonSystemFaultGeneral[46].Q THEN "Unit1.Alarms".systemFaultGeneral[46] := TRUE; END_IF;
END_REGION

REGION Network 52: PFE System Fault General 47
   RUNG wire#powerrail
      I_Contact( "Unit1.ControlNodes".fuse[47] )
      { S7_Templates := "time_type := Time" } "Unit1.Alarms".tonSystemFaultGeneral[47].TON(pt := #DelayTime, et =>)
      S_Coil( "Unit1.Alarms".systemFaultGeneral[47] )
   END_RUNG
   // the same network as SCL:
   "Unit1.Alarms".tonSystemFaultGeneral[47].TON(IN := NOT "Unit1.ControlNodes".fuse[47], PT := #DelayTime);
   IF "Unit1.Alarms".tonSystemFaultGeneral[47].Q THEN "Unit1.Alarms".systemFaultGeneral[47] := TRUE; END_IF;
END_REGION

REGION Network 53: PFE System Fault General 48
   RUNG wire#powerrail
      I_Contact( "Unit1.ControlNodes".fuse[48] )
      { S7_Templates := "time_type := Time" } "Unit1.Alarms".tonSystemFaultGeneral[48].TON(pt := #DelayTime, et =>)
      S_Coil( "Unit1.Alarms".systemFaultGeneral[48] )
   END_RUNG
   // the same network as SCL:
   "Unit1.Alarms".tonSystemFaultGeneral[48].TON(IN := NOT "Unit1.ControlNodes".fuse[48], PT := #DelayTime);
   IF "Unit1.Alarms".tonSystemFaultGeneral[48].Q THEN "Unit1.Alarms".systemFaultGeneral[48] := TRUE; END_IF;
END_REGION

REGION Network 54: PFE System Fault General 49
   RUNG wire#powerrail
      I_Contact( "Unit1.ControlNodes".fuse[49] )
      { S7_Templates := "time_type := Time" } "Unit1.Alarms".tonSystemFaultGeneral[49].TON(pt := #DelayTime, et =>)
      S_Coil( "Unit1.Alarms".systemFaultGeneral[49] )
   END_RUNG
   // the same network as SCL:
   "Unit1.Alarms".tonSystemFaultGeneral[49].TON(IN := NOT "Unit1.ControlNodes".fuse[49], PT := #DelayTime);
   IF "Unit1.Alarms".tonSystemFaultGeneral[49].Q THEN "Unit1.Alarms".systemFaultGeneral[49] := TRUE; END_IF;
END_REGION

REGION Network 55: PFE System Fault General 50
   RUNG wire#powerrail
      I_Contact( "Unit1.ControlNodes".fuse[50] )
      { S7_Templates := "time_type := Time" } "Unit1.Alarms".tonSystemFaultGeneral[50].TON(pt := #DelayTime, et =>)
      S_Coil( "Unit1.Alarms".systemFaultGeneral[50] )
   END_RUNG
   // the same network as SCL:
   "Unit1.Alarms".tonSystemFaultGeneral[50].TON(IN := NOT "Unit1.ControlNodes".fuse[50], PT := #DelayTime);
   IF "Unit1.Alarms".tonSystemFaultGeneral[50].Q THEN "Unit1.Alarms".systemFaultGeneral[50] := TRUE; END_IF;
END_REGION

REGION Network 56: PFE System Fault General 51
   RUNG wire#powerrail
      I_Contact( "Unit1.ControlNodes".fuse[51] )
      { S7_Templates := "time_type := Time" } "Unit1.Alarms".tonSystemFaultGeneral[51].TON(pt := #DelayTime, et =>)
      S_Coil( "Unit1.Alarms".systemFaultGeneral[51] )
   END_RUNG
   // the same network as SCL:
   "Unit1.Alarms".tonSystemFaultGeneral[51].TON(IN := NOT "Unit1.ControlNodes".fuse[51], PT := #DelayTime);
   IF "Unit1.Alarms".tonSystemFaultGeneral[51].Q THEN "Unit1.Alarms".systemFaultGeneral[51] := TRUE; END_IF;
END_REGION

REGION Network 57: PFE System Fault General 52
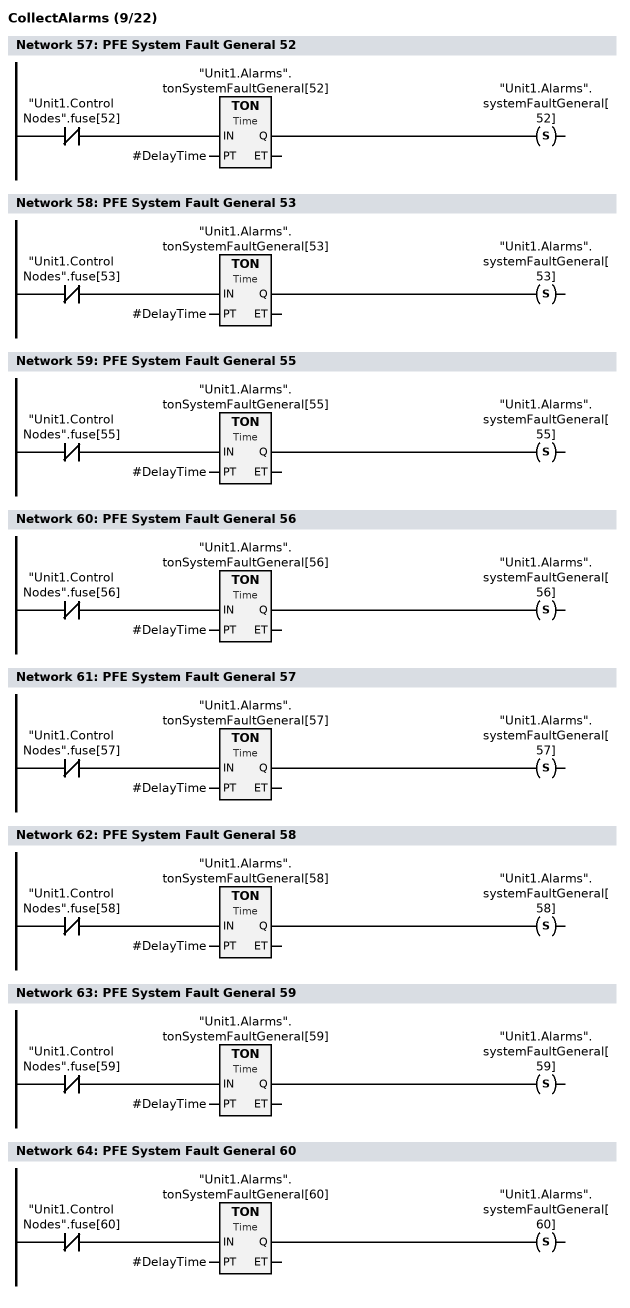
   RUNG wire#powerrail
      I_Contact( "Unit1.ControlNodes".fuse[52] )
      { S7_Templates := "time_type := Time" } "Unit1.Alarms".tonSystemFaultGeneral[52].TON(pt := #DelayTime, et =>)
      S_Coil( "Unit1.Alarms".systemFaultGeneral[52] )
   END_RUNG
   // the same network as SCL:
   "Unit1.Alarms".tonSystemFaultGeneral[52].TON(IN := NOT "Unit1.ControlNodes".fuse[52], PT := #DelayTime);
   IF "Unit1.Alarms".tonSystemFaultGeneral[52].Q THEN "Unit1.Alarms".systemFaultGeneral[52] := TRUE; END_IF;
END_REGION

REGION Network 58: PFE System Fault General 53
   RUNG wire#powerrail
      I_Contact( "Unit1.ControlNodes".fuse[53] )
      { S7_Templates := "time_type := Time" } "Unit1.Alarms".tonSystemFaultGeneral[53].TON(pt := #DelayTime, et =>)
      S_Coil( "Unit1.Alarms".systemFaultGeneral[53] )
   END_RUNG
   // the same network as SCL:
   "Unit1.Alarms".tonSystemFaultGeneral[53].TON(IN := NOT "Unit1.ControlNodes".fuse[53], PT := #DelayTime);
   IF "Unit1.Alarms".tonSystemFaultGeneral[53].Q THEN "Unit1.Alarms".systemFaultGeneral[53] := TRUE; END_IF;
END_REGION

REGION Network 59: PFE System Fault General 55
   RUNG wire#powerrail
      I_Contact( "Unit1.ControlNodes".fuse[55] )
      { S7_Templates := "time_type := Time" } "Unit1.Alarms".tonSystemFaultGeneral[55].TON(pt := #DelayTime, et =>)
      S_Coil( "Unit1.Alarms".systemFaultGeneral[55] )
   END_RUNG
   // the same network as SCL:
   "Unit1.Alarms".tonSystemFaultGeneral[55].TON(IN := NOT "Unit1.ControlNodes".fuse[55], PT := #DelayTime);
   IF "Unit1.Alarms".tonSystemFaultGeneral[55].Q THEN "Unit1.Alarms".systemFaultGeneral[55] := TRUE; END_IF;
END_REGION

REGION Network 60: PFE System Fault General 56
   RUNG wire#powerrail
      I_Contact( "Unit1.ControlNodes".fuse[56] )
      { S7_Templates := "time_type := Time" } "Unit1.Alarms".tonSystemFaultGeneral[56].TON(pt := #DelayTime, et =>)
      S_Coil( "Unit1.Alarms".systemFaultGeneral[56] )
   END_RUNG
   // the same network as SCL:
   "Unit1.Alarms".tonSystemFaultGeneral[56].TON(IN := NOT "Unit1.ControlNodes".fuse[56], PT := #DelayTime);
   IF "Unit1.Alarms".tonSystemFaultGeneral[56].Q THEN "Unit1.Alarms".systemFaultGeneral[56] := TRUE; END_IF;
END_REGION

REGION Network 61: PFE System Fault General 57
   RUNG wire#powerrail
      I_Contact( "Unit1.ControlNodes".fuse[57] )
      { S7_Templates := "time_type := Time" } "Unit1.Alarms".tonSystemFaultGeneral[57].TON(pt := #DelayTime, et =>)
      S_Coil( "Unit1.Alarms".systemFaultGeneral[57] )
   END_RUNG
   // the same network as SCL:
   "Unit1.Alarms".tonSystemFaultGeneral[57].TON(IN := NOT "Unit1.ControlNodes".fuse[57], PT := #DelayTime);
   IF "Unit1.Alarms".tonSystemFaultGeneral[57].Q THEN "Unit1.Alarms".systemFaultGeneral[57] := TRUE; END_IF;
END_REGION

REGION Network 62: PFE System Fault General 58
   RUNG wire#powerrail
      I_Contact( "Unit1.ControlNodes".fuse[58] )
      { S7_Templates := "time_type := Time" } "Unit1.Alarms".tonSystemFaultGeneral[58].TON(pt := #DelayTime, et =>)
      S_Coil( "Unit1.Alarms".systemFaultGeneral[58] )
   END_RUNG
   // the same network as SCL:
   "Unit1.Alarms".tonSystemFaultGeneral[58].TON(IN := NOT "Unit1.ControlNodes".fuse[58], PT := #DelayTime);
   IF "Unit1.Alarms".tonSystemFaultGeneral[58].Q THEN "Unit1.Alarms".systemFaultGeneral[58] := TRUE; END_IF;
END_REGION

REGION Network 63: PFE System Fault General 59
   RUNG wire#powerrail
      I_Contact( "Unit1.ControlNodes".fuse[59] )
      { S7_Templates := "time_type := Time" } "Unit1.Alarms".tonSystemFaultGeneral[59].TON(pt := #DelayTime, et =>)
      S_Coil( "Unit1.Alarms".systemFaultGeneral[59] )
   END_RUNG
   // the same network as SCL:
   "Unit1.Alarms".tonSystemFaultGeneral[59].TON(IN := NOT "Unit1.ControlNodes".fuse[59], PT := #DelayTime);
   IF "Unit1.Alarms".tonSystemFaultGeneral[59].Q THEN "Unit1.Alarms".systemFaultGeneral[59] := TRUE; END_IF;
END_REGION

REGION Network 64: PFE System Fault General 60
   RUNG wire#powerrail
      I_Contact( "Unit1.ControlNodes".fuse[60] )
      { S7_Templates := "time_type := Time" } "Unit1.Alarms".tonSystemFaultGeneral[60].TON(pt := #DelayTime, et =>)
      S_Coil( "Unit1.Alarms".systemFaultGeneral[60] )
   END_RUNG
   // the same network as SCL:
   "Unit1.Alarms".tonSystemFaultGeneral[60].TON(IN := NOT "Unit1.ControlNodes".fuse[60], PT := #DelayTime);
   IF "Unit1.Alarms".tonSystemFaultGeneral[60].Q THEN "Unit1.Alarms".systemFaultGeneral[60] := TRUE; END_IF;
END_REGION

REGION Network 65: PFE System Fault General 61
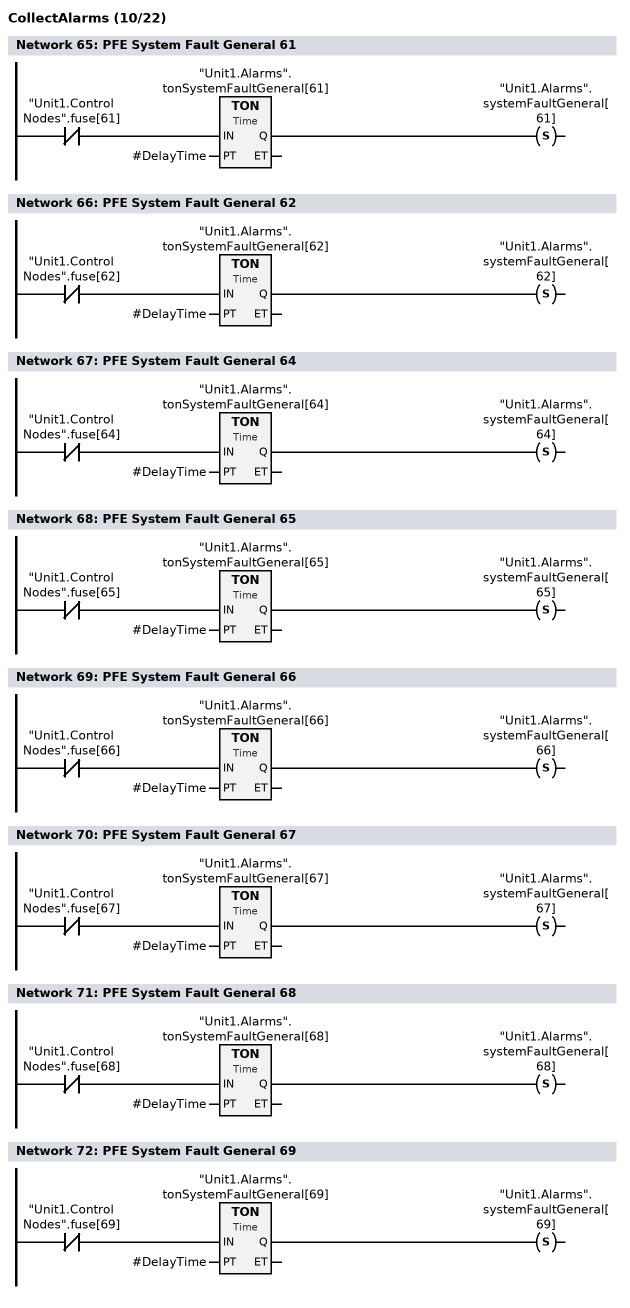
   RUNG wire#powerrail
      I_Contact( "Unit1.ControlNodes".fuse[61] )
      { S7_Templates := "time_type := Time" } "Unit1.Alarms".tonSystemFaultGeneral[61].TON(pt := #DelayTime, et =>)
      S_Coil( "Unit1.Alarms".systemFaultGeneral[61] )
   END_RUNG
   // the same network as SCL:
   "Unit1.Alarms".tonSystemFaultGeneral[61].TON(IN := NOT "Unit1.ControlNodes".fuse[61], PT := #DelayTime);
   IF "Unit1.Alarms".tonSystemFaultGeneral[61].Q THEN "Unit1.Alarms".systemFaultGeneral[61] := TRUE; END_IF;
END_REGION

REGION Network 66: PFE System Fault General 62
   RUNG wire#powerrail
      I_Contact( "Unit1.ControlNodes".fuse[62] )
      { S7_Templates := "time_type := Time" } "Unit1.Alarms".tonSystemFaultGeneral[62].TON(pt := #DelayTime, et =>)
      S_Coil( "Unit1.Alarms".systemFaultGeneral[62] )
   END_RUNG
   // the same network as SCL:
   "Unit1.Alarms".tonSystemFaultGeneral[62].TON(IN := NOT "Unit1.ControlNodes".fuse[62], PT := #DelayTime);
   IF "Unit1.Alarms".tonSystemFaultGeneral[62].Q THEN "Unit1.Alarms".systemFaultGeneral[62] := TRUE; END_IF;
END_REGION

REGION Network 67: PFE System Fault General 64
   RUNG wire#powerrail
      I_Contact( "Unit1.ControlNodes".fuse[64] )
      { S7_Templates := "time_type := Time" } "Unit1.Alarms".tonSystemFaultGeneral[64].TON(pt := #DelayTime, et =>)
      S_Coil( "Unit1.Alarms".systemFaultGeneral[64] )
   END_RUNG
   // the same network as SCL:
   "Unit1.Alarms".tonSystemFaultGeneral[64].TON(IN := NOT "Unit1.ControlNodes".fuse[64], PT := #DelayTime);
   IF "Unit1.Alarms".tonSystemFaultGeneral[64].Q THEN "Unit1.Alarms".systemFaultGeneral[64] := TRUE; END_IF;
END_REGION

REGION Network 68: PFE System Fault General 65
   RUNG wire#powerrail
      I_Contact( "Unit1.ControlNodes".fuse[65] )
      { S7_Templates := "time_type := Time" } "Unit1.Alarms".tonSystemFaultGeneral[65].TON(pt := #DelayTime, et =>)
      S_Coil( "Unit1.Alarms".systemFaultGeneral[65] )
   END_RUNG
   // the same network as SCL:
   "Unit1.Alarms".tonSystemFaultGeneral[65].TON(IN := NOT "Unit1.ControlNodes".fuse[65], PT := #DelayTime);
   IF "Unit1.Alarms".tonSystemFaultGeneral[65].Q THEN "Unit1.Alarms".systemFaultGeneral[65] := TRUE; END_IF;
END_REGION

REGION Network 69: PFE System Fault General 66
   RUNG wire#powerrail
      I_Contact( "Unit1.ControlNodes".fuse[66] )
      { S7_Templates := "time_type := Time" } "Unit1.Alarms".tonSystemFaultGeneral[66].TON(pt := #DelayTime, et =>)
      S_Coil( "Unit1.Alarms".systemFaultGeneral[66] )
   END_RUNG
   // the same network as SCL:
   "Unit1.Alarms".tonSystemFaultGeneral[66].TON(IN := NOT "Unit1.ControlNodes".fuse[66], PT := #DelayTime);
   IF "Unit1.Alarms".tonSystemFaultGeneral[66].Q THEN "Unit1.Alarms".systemFaultGeneral[66] := TRUE; END_IF;
END_REGION

REGION Network 70: PFE System Fault General 67
   RUNG wire#powerrail
      I_Contact( "Unit1.ControlNodes".fuse[67] )
      { S7_Templates := "time_type := Time" } "Unit1.Alarms".tonSystemFaultGeneral[67].TON(pt := #DelayTime, et =>)
      S_Coil( "Unit1.Alarms".systemFaultGeneral[67] )
   END_RUNG
   // the same network as SCL:
   "Unit1.Alarms".tonSystemFaultGeneral[67].TON(IN := NOT "Unit1.ControlNodes".fuse[67], PT := #DelayTime);
   IF "Unit1.Alarms".tonSystemFaultGeneral[67].Q THEN "Unit1.Alarms".systemFaultGeneral[67] := TRUE; END_IF;
END_REGION

REGION Network 71: PFE System Fault General 68
   RUNG wire#powerrail
      I_Contact( "Unit1.ControlNodes".fuse[68] )
      { S7_Templates := "time_type := Time" } "Unit1.Alarms".tonSystemFaultGeneral[68].TON(pt := #DelayTime, et =>)
      S_Coil( "Unit1.Alarms".systemFaultGeneral[68] )
   END_RUNG
   // the same network as SCL:
   "Unit1.Alarms".tonSystemFaultGeneral[68].TON(IN := NOT "Unit1.ControlNodes".fuse[68], PT := #DelayTime);
   IF "Unit1.Alarms".tonSystemFaultGeneral[68].Q THEN "Unit1.Alarms".systemFaultGeneral[68] := TRUE; END_IF;
END_REGION

REGION Network 72: PFE System Fault General 69
   RUNG wire#powerrail
      I_Contact( "Unit1.ControlNodes".fuse[69] )
      { S7_Templates := "time_type := Time" } "Unit1.Alarms".tonSystemFaultGeneral[69].TON(pt := #DelayTime, et =>)
      S_Coil( "Unit1.Alarms".systemFaultGeneral[69] )
   END_RUNG
   // the same network as SCL:
   "Unit1.Alarms".tonSystemFaultGeneral[69].TON(IN := NOT "Unit1.ControlNodes".fuse[69], PT := #DelayTime);
   IF "Unit1.Alarms".tonSystemFaultGeneral[69].Q THEN "Unit1.Alarms".systemFaultGeneral[69] := TRUE; END_IF;
END_REGION

REGION Network 73: PFE System Fault General 70
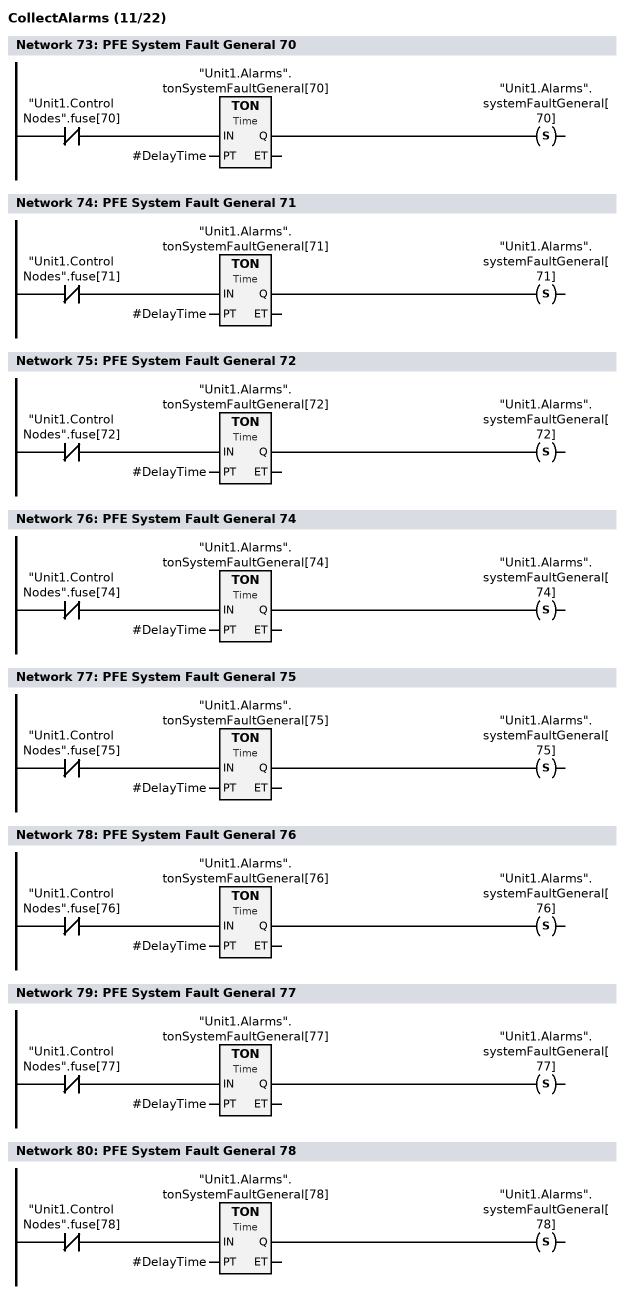
   RUNG wire#powerrail
      I_Contact( "Unit1.ControlNodes".fuse[70] )
      { S7_Templates := "time_type := Time" } "Unit1.Alarms".tonSystemFaultGeneral[70].TON(pt := #DelayTime, et =>)
      S_Coil( "Unit1.Alarms".systemFaultGeneral[70] )
   END_RUNG
   // the same network as SCL:
   "Unit1.Alarms".tonSystemFaultGeneral[70].TON(IN := NOT "Unit1.ControlNodes".fuse[70], PT := #DelayTime);
   IF "Unit1.Alarms".tonSystemFaultGeneral[70].Q THEN "Unit1.Alarms".systemFaultGeneral[70] := TRUE; END_IF;
END_REGION

REGION Network 74: PFE System Fault General 71
   RUNG wire#powerrail
      I_Contact( "Unit1.ControlNodes".fuse[71] )
      { S7_Templates := "time_type := Time" } "Unit1.Alarms".tonSystemFaultGeneral[71].TON(pt := #DelayTime, et =>)
      S_Coil( "Unit1.Alarms".systemFaultGeneral[71] )
   END_RUNG
   // the same network as SCL:
   "Unit1.Alarms".tonSystemFaultGeneral[71].TON(IN := NOT "Unit1.ControlNodes".fuse[71], PT := #DelayTime);
   IF "Unit1.Alarms".tonSystemFaultGeneral[71].Q THEN "Unit1.Alarms".systemFaultGeneral[71] := TRUE; END_IF;
END_REGION

REGION Network 75: PFE System Fault General 72
   RUNG wire#powerrail
      I_Contact( "Unit1.ControlNodes".fuse[72] )
      { S7_Templates := "time_type := Time" } "Unit1.Alarms".tonSystemFaultGeneral[72].TON(pt := #DelayTime, et =>)
      S_Coil( "Unit1.Alarms".systemFaultGeneral[72] )
   END_RUNG
   // the same network as SCL:
   "Unit1.Alarms".tonSystemFaultGeneral[72].TON(IN := NOT "Unit1.ControlNodes".fuse[72], PT := #DelayTime);
   IF "Unit1.Alarms".tonSystemFaultGeneral[72].Q THEN "Unit1.Alarms".systemFaultGeneral[72] := TRUE; END_IF;
END_REGION

REGION Network 76: PFE System Fault General 74
   RUNG wire#powerrail
      I_Contact( "Unit1.ControlNodes".fuse[74] )
      { S7_Templates := "time_type := Time" } "Unit1.Alarms".tonSystemFaultGeneral[74].TON(pt := #DelayTime, et =>)
      S_Coil( "Unit1.Alarms".systemFaultGeneral[74] )
   END_RUNG
   // the same network as SCL:
   "Unit1.Alarms".tonSystemFaultGeneral[74].TON(IN := NOT "Unit1.ControlNodes".fuse[74], PT := #DelayTime);
   IF "Unit1.Alarms".tonSystemFaultGeneral[74].Q THEN "Unit1.Alarms".systemFaultGeneral[74] := TRUE; END_IF;
END_REGION

REGION Network 77: PFE System Fault General 75
   RUNG wire#powerrail
      I_Contact( "Unit1.ControlNodes".fuse[75] )
      { S7_Templates := "time_type := Time" } "Unit1.Alarms".tonSystemFaultGeneral[75].TON(pt := #DelayTime, et =>)
      S_Coil( "Unit1.Alarms".systemFaultGeneral[75] )
   END_RUNG
   // the same network as SCL:
   "Unit1.Alarms".tonSystemFaultGeneral[75].TON(IN := NOT "Unit1.ControlNodes".fuse[75], PT := #DelayTime);
   IF "Unit1.Alarms".tonSystemFaultGeneral[75].Q THEN "Unit1.Alarms".systemFaultGeneral[75] := TRUE; END_IF;
END_REGION

REGION Network 78: PFE System Fault General 76
   RUNG wire#powerrail
      I_Contact( "Unit1.ControlNodes".fuse[76] )
      { S7_Templates := "time_type := Time" } "Unit1.Alarms".tonSystemFaultGeneral[76].TON(pt := #DelayTime, et =>)
      S_Coil( "Unit1.Alarms".systemFaultGeneral[76] )
   END_RUNG
   // the same network as SCL:
   "Unit1.Alarms".tonSystemFaultGeneral[76].TON(IN := NOT "Unit1.ControlNodes".fuse[76], PT := #DelayTime);
   IF "Unit1.Alarms".tonSystemFaultGeneral[76].Q THEN "Unit1.Alarms".systemFaultGeneral[76] := TRUE; END_IF;
END_REGION

REGION Network 79: PFE System Fault General 77
   RUNG wire#powerrail
      I_Contact( "Unit1.ControlNodes".fuse[77] )
      { S7_Templates := "time_type := Time" } "Unit1.Alarms".tonSystemFaultGeneral[77].TON(pt := #DelayTime, et =>)
      S_Coil( "Unit1.Alarms".systemFaultGeneral[77] )
   END_RUNG
   // the same network as SCL:
   "Unit1.Alarms".tonSystemFaultGeneral[77].TON(IN := NOT "Unit1.ControlNodes".fuse[77], PT := #DelayTime);
   IF "Unit1.Alarms".tonSystemFaultGeneral[77].Q THEN "Unit1.Alarms".systemFaultGeneral[77] := TRUE; END_IF;
END_REGION

REGION Network 80: PFE System Fault General 78
   RUNG wire#powerrail
      I_Contact( "Unit1.ControlNodes".fuse[78] )
      { S7_Templates := "time_type := Time" } "Unit1.Alarms".tonSystemFaultGeneral[78].TON(pt := #DelayTime, et =>)
      S_Coil( "Unit1.Alarms".systemFaultGeneral[78] )
   END_RUNG
   // the same network as SCL:
   "Unit1.Alarms".tonSystemFaultGeneral[78].TON(IN := NOT "Unit1.ControlNodes".fuse[78], PT := #DelayTime);
   IF "Unit1.Alarms".tonSystemFaultGeneral[78].Q THEN "Unit1.Alarms".systemFaultGeneral[78] := TRUE; END_IF;
END_REGION

REGION Network 81: PFE System Fault General 80
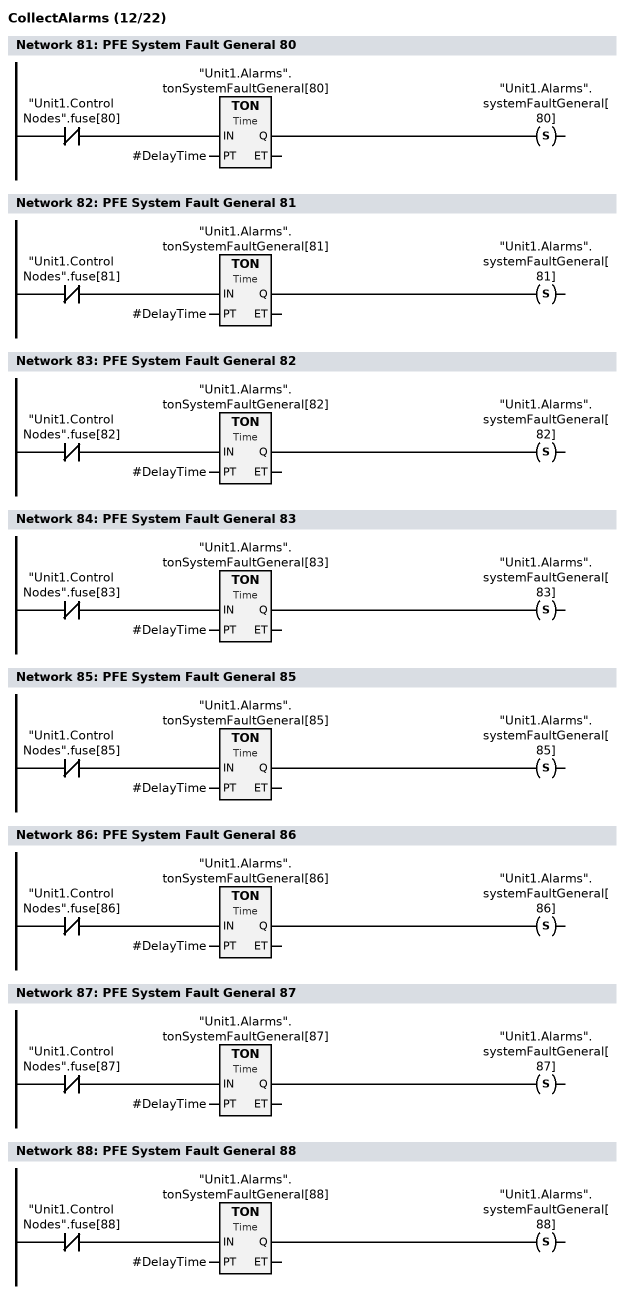
   RUNG wire#powerrail
      I_Contact( "Unit1.ControlNodes".fuse[80] )
      { S7_Templates := "time_type := Time" } "Unit1.Alarms".tonSystemFaultGeneral[80].TON(pt := #DelayTime, et =>)
      S_Coil( "Unit1.Alarms".systemFaultGeneral[80] )
   END_RUNG
   // the same network as SCL:
   "Unit1.Alarms".tonSystemFaultGeneral[80].TON(IN := NOT "Unit1.ControlNodes".fuse[80], PT := #DelayTime);
   IF "Unit1.Alarms".tonSystemFaultGeneral[80].Q THEN "Unit1.Alarms".systemFaultGeneral[80] := TRUE; END_IF;
END_REGION

REGION Network 82: PFE System Fault General 81
   RUNG wire#powerrail
      I_Contact( "Unit1.ControlNodes".fuse[81] )
      { S7_Templates := "time_type := Time" } "Unit1.Alarms".tonSystemFaultGeneral[81].TON(pt := #DelayTime, et =>)
      S_Coil( "Unit1.Alarms".systemFaultGeneral[81] )
   END_RUNG
   // the same network as SCL:
   "Unit1.Alarms".tonSystemFaultGeneral[81].TON(IN := NOT "Unit1.ControlNodes".fuse[81], PT := #DelayTime);
   IF "Unit1.Alarms".tonSystemFaultGeneral[81].Q THEN "Unit1.Alarms".systemFaultGeneral[81] := TRUE; END_IF;
END_REGION

REGION Network 83: PFE System Fault General 82
   RUNG wire#powerrail
      I_Contact( "Unit1.ControlNodes".fuse[82] )
      { S7_Templates := "time_type := Time" } "Unit1.Alarms".tonSystemFaultGeneral[82].TON(pt := #DelayTime, et =>)
      S_Coil( "Unit1.Alarms".systemFaultGeneral[82] )
   END_RUNG
   // the same network as SCL:
   "Unit1.Alarms".tonSystemFaultGeneral[82].TON(IN := NOT "Unit1.ControlNodes".fuse[82], PT := #DelayTime);
   IF "Unit1.Alarms".tonSystemFaultGeneral[82].Q THEN "Unit1.Alarms".systemFaultGeneral[82] := TRUE; END_IF;
END_REGION

REGION Network 84: PFE System Fault General 83
   RUNG wire#powerrail
      I_Contact( "Unit1.ControlNodes".fuse[83] )
      { S7_Templates := "time_type := Time" } "Unit1.Alarms".tonSystemFaultGeneral[83].TON(pt := #DelayTime, et =>)
      S_Coil( "Unit1.Alarms".systemFaultGeneral[83] )
   END_RUNG
   // the same network as SCL:
   "Unit1.Alarms".tonSystemFaultGeneral[83].TON(IN := NOT "Unit1.ControlNodes".fuse[83], PT := #DelayTime);
   IF "Unit1.Alarms".tonSystemFaultGeneral[83].Q THEN "Unit1.Alarms".systemFaultGeneral[83] := TRUE; END_IF;
END_REGION

REGION Network 85: PFE System Fault General 85
   RUNG wire#powerrail
      I_Contact( "Unit1.ControlNodes".fuse[85] )
      { S7_Templates := "time_type := Time" } "Unit1.Alarms".tonSystemFaultGeneral[85].TON(pt := #DelayTime, et =>)
      S_Coil( "Unit1.Alarms".systemFaultGeneral[85] )
   END_RUNG
   // the same network as SCL:
   "Unit1.Alarms".tonSystemFaultGeneral[85].TON(IN := NOT "Unit1.ControlNodes".fuse[85], PT := #DelayTime);
   IF "Unit1.Alarms".tonSystemFaultGeneral[85].Q THEN "Unit1.Alarms".systemFaultGeneral[85] := TRUE; END_IF;
END_REGION

REGION Network 86: PFE System Fault General 86
   RUNG wire#powerrail
      I_Contact( "Unit1.ControlNodes".fuse[86] )
      { S7_Templates := "time_type := Time" } "Unit1.Alarms".tonSystemFaultGeneral[86].TON(pt := #DelayTime, et =>)
      S_Coil( "Unit1.Alarms".systemFaultGeneral[86] )
   END_RUNG
   // the same network as SCL:
   "Unit1.Alarms".tonSystemFaultGeneral[86].TON(IN := NOT "Unit1.ControlNodes".fuse[86], PT := #DelayTime);
   IF "Unit1.Alarms".tonSystemFaultGeneral[86].Q THEN "Unit1.Alarms".systemFaultGeneral[86] := TRUE; END_IF;
END_REGION

REGION Network 87: PFE System Fault General 87
   RUNG wire#powerrail
      I_Contact( "Unit1.ControlNodes".fuse[87] )
      { S7_Templates := "time_type := Time" } "Unit1.Alarms".tonSystemFaultGeneral[87].TON(pt := #DelayTime, et =>)
      S_Coil( "Unit1.Alarms".systemFaultGeneral[87] )
   END_RUNG
   // the same network as SCL:
   "Unit1.Alarms".tonSystemFaultGeneral[87].TON(IN := NOT "Unit1.ControlNodes".fuse[87], PT := #DelayTime);
   IF "Unit1.Alarms".tonSystemFaultGeneral[87].Q THEN "Unit1.Alarms".systemFaultGeneral[87] := TRUE; END_IF;
END_REGION

REGION Network 88: PFE System Fault General 88
   RUNG wire#powerrail
      I_Contact( "Unit1.ControlNodes".fuse[88] )
      { S7_Templates := "time_type := Time" } "Unit1.Alarms".tonSystemFaultGeneral[88].TON(pt := #DelayTime, et =>)
      S_Coil( "Unit1.Alarms".systemFaultGeneral[88] )
   END_RUNG
   // the same network as SCL:
   "Unit1.Alarms".tonSystemFaultGeneral[88].TON(IN := NOT "Unit1.ControlNodes".fuse[88], PT := #DelayTime);
   IF "Unit1.Alarms".tonSystemFaultGeneral[88].Q THEN "Unit1.Alarms".systemFaultGeneral[88] := TRUE; END_IF;
END_REGION

REGION Network 89: PFE System Fault General 89
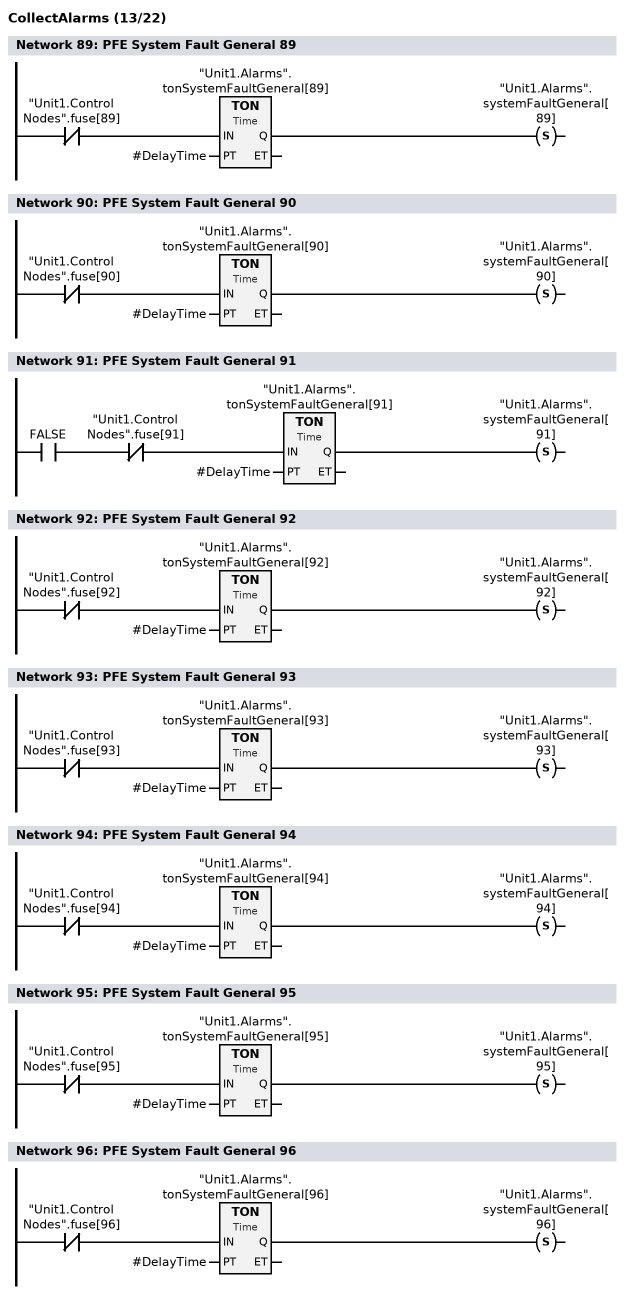
   RUNG wire#powerrail
      I_Contact( "Unit1.ControlNodes".fuse[89] )
      { S7_Templates := "time_type := Time" } "Unit1.Alarms".tonSystemFaultGeneral[89].TON(pt := #DelayTime, et =>)
      S_Coil( "Unit1.Alarms".systemFaultGeneral[89] )
   END_RUNG
   // the same network as SCL:
   "Unit1.Alarms".tonSystemFaultGeneral[89].TON(IN := NOT "Unit1.ControlNodes".fuse[89], PT := #DelayTime);
   IF "Unit1.Alarms".tonSystemFaultGeneral[89].Q THEN "Unit1.Alarms".systemFaultGeneral[89] := TRUE; END_IF;
END_REGION

REGION Network 90: PFE System Fault General 90
   RUNG wire#powerrail
      I_Contact( "Unit1.ControlNodes".fuse[90] )
      { S7_Templates := "time_type := Time" } "Unit1.Alarms".tonSystemFaultGeneral[90].TON(pt := #DelayTime, et =>)
      S_Coil( "Unit1.Alarms".systemFaultGeneral[90] )
   END_RUNG
   // the same network as SCL:
   "Unit1.Alarms".tonSystemFaultGeneral[90].TON(IN := NOT "Unit1.ControlNodes".fuse[90], PT := #DelayTime);
   IF "Unit1.Alarms".tonSystemFaultGeneral[90].Q THEN "Unit1.Alarms".systemFaultGeneral[90] := TRUE; END_IF;
END_REGION

REGION Network 91: PFE System Fault General 91
   RUNG wire#powerrail
      Contact( FALSE )
      I_Contact( "Unit1.ControlNodes".fuse[91] )
      { S7_Templates := "time_type := Time" } "Unit1.Alarms".tonSystemFaultGeneral[91].TON(pt := #DelayTime, et =>)
      S_Coil( "Unit1.Alarms".systemFaultGeneral[91] )
   END_RUNG
   // the same network as SCL:
   "Unit1.Alarms".tonSystemFaultGeneral[91].TON(IN := FALSE AND NOT "Unit1.ControlNodes".fuse[91],
                           PT := #DelayTime);
   IF "Unit1.Alarms".tonSystemFaultGeneral[91].Q THEN "Unit1.Alarms".systemFaultGeneral[91] := TRUE; END_IF;
END_REGION

REGION Network 92: PFE System Fault General 92
   RUNG wire#powerrail
      I_Contact( "Unit1.ControlNodes".fuse[92] )
      { S7_Templates := "time_type := Time" } "Unit1.Alarms".tonSystemFaultGeneral[92].TON(pt := #DelayTime, et =>)
      S_Coil( "Unit1.Alarms".systemFaultGeneral[92] )
   END_RUNG
   // the same network as SCL:
   "Unit1.Alarms".tonSystemFaultGeneral[92].TON(IN := NOT "Unit1.ControlNodes".fuse[92], PT := #DelayTime);
   IF "Unit1.Alarms".tonSystemFaultGeneral[92].Q THEN "Unit1.Alarms".systemFaultGeneral[92] := TRUE; END_IF;
END_REGION

REGION Network 93: PFE System Fault General 93
   RUNG wire#powerrail
      I_Contact( "Unit1.ControlNodes".fuse[93] )
      { S7_Templates := "time_type := Time" } "Unit1.Alarms".tonSystemFaultGeneral[93].TON(pt := #DelayTime, et =>)
      S_Coil( "Unit1.Alarms".systemFaultGeneral[93] )
   END_RUNG
   // the same network as SCL:
   "Unit1.Alarms".tonSystemFaultGeneral[93].TON(IN := NOT "Unit1.ControlNodes".fuse[93], PT := #DelayTime);
   IF "Unit1.Alarms".tonSystemFaultGeneral[93].Q THEN "Unit1.Alarms".systemFaultGeneral[93] := TRUE; END_IF;
END_REGION

REGION Network 94: PFE System Fault General 94
   RUNG wire#powerrail
      I_Contact( "Unit1.ControlNodes".fuse[94] )
      { S7_Templates := "time_type := Time" } "Unit1.Alarms".tonSystemFaultGeneral[94].TON(pt := #DelayTime, et =>)
      S_Coil( "Unit1.Alarms".systemFaultGeneral[94] )
   END_RUNG
   // the same network as SCL:
   "Unit1.Alarms".tonSystemFaultGeneral[94].TON(IN := NOT "Unit1.ControlNodes".fuse[94], PT := #DelayTime);
   IF "Unit1.Alarms".tonSystemFaultGeneral[94].Q THEN "Unit1.Alarms".systemFaultGeneral[94] := TRUE; END_IF;
END_REGION

REGION Network 95: PFE System Fault General 95
   RUNG wire#powerrail
      I_Contact( "Unit1.ControlNodes".fuse[95] )
      { S7_Templates := "time_type := Time" } "Unit1.Alarms".tonSystemFaultGeneral[95].TON(pt := #DelayTime, et =>)
      S_Coil( "Unit1.Alarms".systemFaultGeneral[95] )
   END_RUNG
   // the same network as SCL:
   "Unit1.Alarms".tonSystemFaultGeneral[95].TON(IN := NOT "Unit1.ControlNodes".fuse[95], PT := #DelayTime);
   IF "Unit1.Alarms".tonSystemFaultGeneral[95].Q THEN "Unit1.Alarms".systemFaultGeneral[95] := TRUE; END_IF;
END_REGION

REGION Network 96: PFE System Fault General 96
   RUNG wire#powerrail
      I_Contact( "Unit1.ControlNodes".fuse[96] )
      { S7_Templates := "time_type := Time" } "Unit1.Alarms".tonSystemFaultGeneral[96].TON(pt := #DelayTime, et =>)
      S_Coil( "Unit1.Alarms".systemFaultGeneral[96] )
   END_RUNG
   // the same network as SCL:
   "Unit1.Alarms".tonSystemFaultGeneral[96].TON(IN := NOT "Unit1.ControlNodes".fuse[96], PT := #DelayTime);
   IF "Unit1.Alarms".tonSystemFaultGeneral[96].Q THEN "Unit1.Alarms".systemFaultGeneral[96] := TRUE; END_IF;
END_REGION

REGION Network 97: PFE System Fault General 97
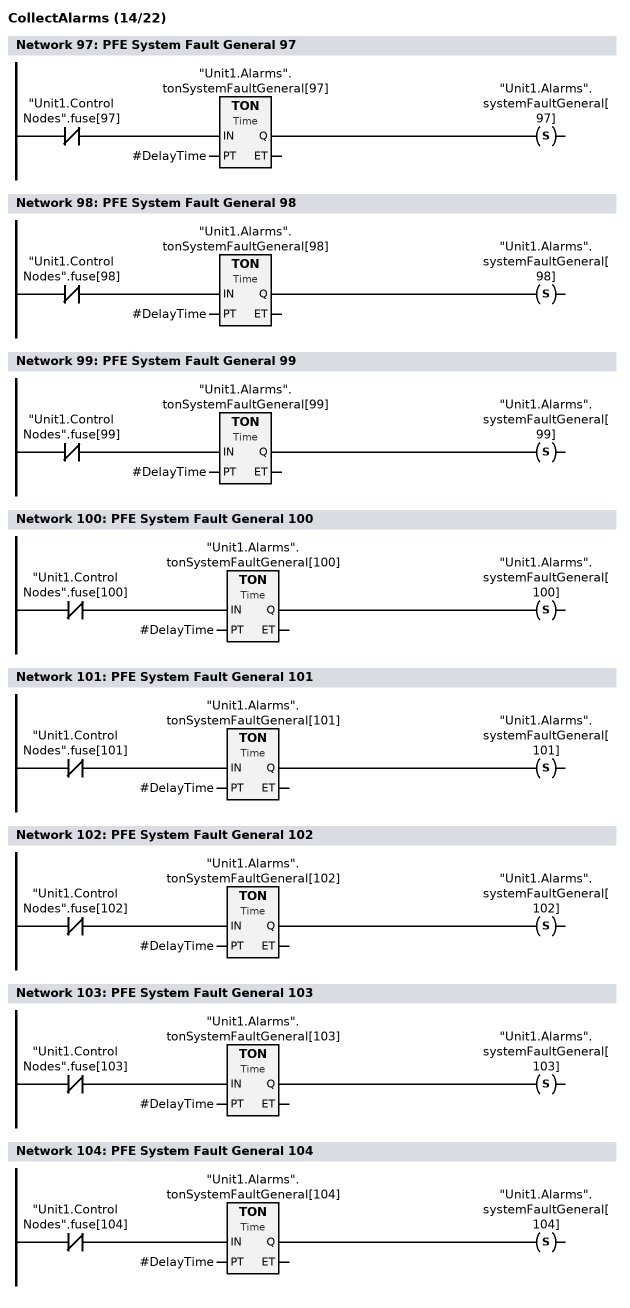
   RUNG wire#powerrail
      I_Contact( "Unit1.ControlNodes".fuse[97] )
      { S7_Templates := "time_type := Time" } "Unit1.Alarms".tonSystemFaultGeneral[97].TON(pt := #DelayTime, et =>)
      S_Coil( "Unit1.Alarms".systemFaultGeneral[97] )
   END_RUNG
   // the same network as SCL:
   "Unit1.Alarms".tonSystemFaultGeneral[97].TON(IN := NOT "Unit1.ControlNodes".fuse[97], PT := #DelayTime);
   IF "Unit1.Alarms".tonSystemFaultGeneral[97].Q THEN "Unit1.Alarms".systemFaultGeneral[97] := TRUE; END_IF;
END_REGION

REGION Network 98: PFE System Fault General 98
   RUNG wire#powerrail
      I_Contact( "Unit1.ControlNodes".fuse[98] )
      { S7_Templates := "time_type := Time" } "Unit1.Alarms".tonSystemFaultGeneral[98].TON(pt := #DelayTime, et =>)
      S_Coil( "Unit1.Alarms".systemFaultGeneral[98] )
   END_RUNG
   // the same network as SCL:
   "Unit1.Alarms".tonSystemFaultGeneral[98].TON(IN := NOT "Unit1.ControlNodes".fuse[98], PT := #DelayTime);
   IF "Unit1.Alarms".tonSystemFaultGeneral[98].Q THEN "Unit1.Alarms".systemFaultGeneral[98] := TRUE; END_IF;
END_REGION

REGION Network 99: PFE System Fault General 99
   RUNG wire#powerrail
      I_Contact( "Unit1.ControlNodes".fuse[99] )
      { S7_Templates := "time_type := Time" } "Unit1.Alarms".tonSystemFaultGeneral[99].TON(pt := #DelayTime, et =>)
      S_Coil( "Unit1.Alarms".systemFaultGeneral[99] )
   END_RUNG
   // the same network as SCL:
   "Unit1.Alarms".tonSystemFaultGeneral[99].TON(IN := NOT "Unit1.ControlNodes".fuse[99], PT := #DelayTime);
   IF "Unit1.Alarms".tonSystemFaultGeneral[99].Q THEN "Unit1.Alarms".systemFaultGeneral[99] := TRUE; END_IF;
END_REGION

REGION Network 100: PFE System Fault General 100
   RUNG wire#powerrail
      I_Contact( "Unit1.ControlNodes".fuse[100] )
      { S7_Templates := "time_type := Time" } "Unit1.Alarms".tonSystemFaultGeneral[100].TON(pt := #DelayTime, et =>)
      S_Coil( "Unit1.Alarms".systemFaultGeneral[100] )
   END_RUNG
   // the same network as SCL:
   "Unit1.Alarms".tonSystemFaultGeneral[100].TON(IN := NOT "Unit1.ControlNodes".fuse[100], PT := #DelayTime);
   IF "Unit1.Alarms".tonSystemFaultGeneral[100].Q THEN
       "Unit1.Alarms".systemFaultGeneral[100] := TRUE;
   END_IF;
END_REGION

REGION Network 101: PFE System Fault General 101
   RUNG wire#powerrail
      I_Contact( "Unit1.ControlNodes".fuse[101] )
      { S7_Templates := "time_type := Time" } "Unit1.Alarms".tonSystemFaultGeneral[101].TON(pt := #DelayTime, et =>)
      S_Coil( "Unit1.Alarms".systemFaultGeneral[101] )
   END_RUNG
   // the same network as SCL:
   "Unit1.Alarms".tonSystemFaultGeneral[101].TON(IN := NOT "Unit1.ControlNodes".fuse[101], PT := #DelayTime);
   IF "Unit1.Alarms".tonSystemFaultGeneral[101].Q THEN
       "Unit1.Alarms".systemFaultGeneral[101] := TRUE;
   END_IF;
END_REGION

REGION Network 102: PFE System Fault General 102
   RUNG wire#powerrail
      I_Contact( "Unit1.ControlNodes".fuse[102] )
      { S7_Templates := "time_type := Time" } "Unit1.Alarms".tonSystemFaultGeneral[102].TON(pt := #DelayTime, et =>)
      S_Coil( "Unit1.Alarms".systemFaultGeneral[102] )
   END_RUNG
   // the same network as SCL:
   "Unit1.Alarms".tonSystemFaultGeneral[102].TON(IN := NOT "Unit1.ControlNodes".fuse[102], PT := #DelayTime);
   IF "Unit1.Alarms".tonSystemFaultGeneral[102].Q THEN
       "Unit1.Alarms".systemFaultGeneral[102] := TRUE;
   END_IF;
END_REGION

REGION Network 103: PFE System Fault General 103
   RUNG wire#powerrail
      I_Contact( "Unit1.ControlNodes".fuse[103] )
      { S7_Templates := "time_type := Time" } "Unit1.Alarms".tonSystemFaultGeneral[103].TON(pt := #DelayTime, et =>)
      S_Coil( "Unit1.Alarms".systemFaultGeneral[103] )
   END_RUNG
   // the same network as SCL:
   "Unit1.Alarms".tonSystemFaultGeneral[103].TON(IN := NOT "Unit1.ControlNodes".fuse[103], PT := #DelayTime);
   IF "Unit1.Alarms".tonSystemFaultGeneral[103].Q THEN
       "Unit1.Alarms".systemFaultGeneral[103] := TRUE;
   END_IF;
END_REGION

REGION Network 104: PFE System Fault General 104
   RUNG wire#powerrail
      I_Contact( "Unit1.ControlNodes".fuse[104] )
      { S7_Templates := "time_type := Time" } "Unit1.Alarms".tonSystemFaultGeneral[104].TON(pt := #DelayTime, et =>)
      S_Coil( "Unit1.Alarms".systemFaultGeneral[104] )
   END_RUNG
   // the same network as SCL:
   "Unit1.Alarms".tonSystemFaultGeneral[104].TON(IN := NOT "Unit1.ControlNodes".fuse[104], PT := #DelayTime);
   IF "Unit1.Alarms".tonSystemFaultGeneral[104].Q THEN
       "Unit1.Alarms".systemFaultGeneral[104] := TRUE;
   END_IF;
END_REGION

REGION Network 105: PFE System Fault General 105
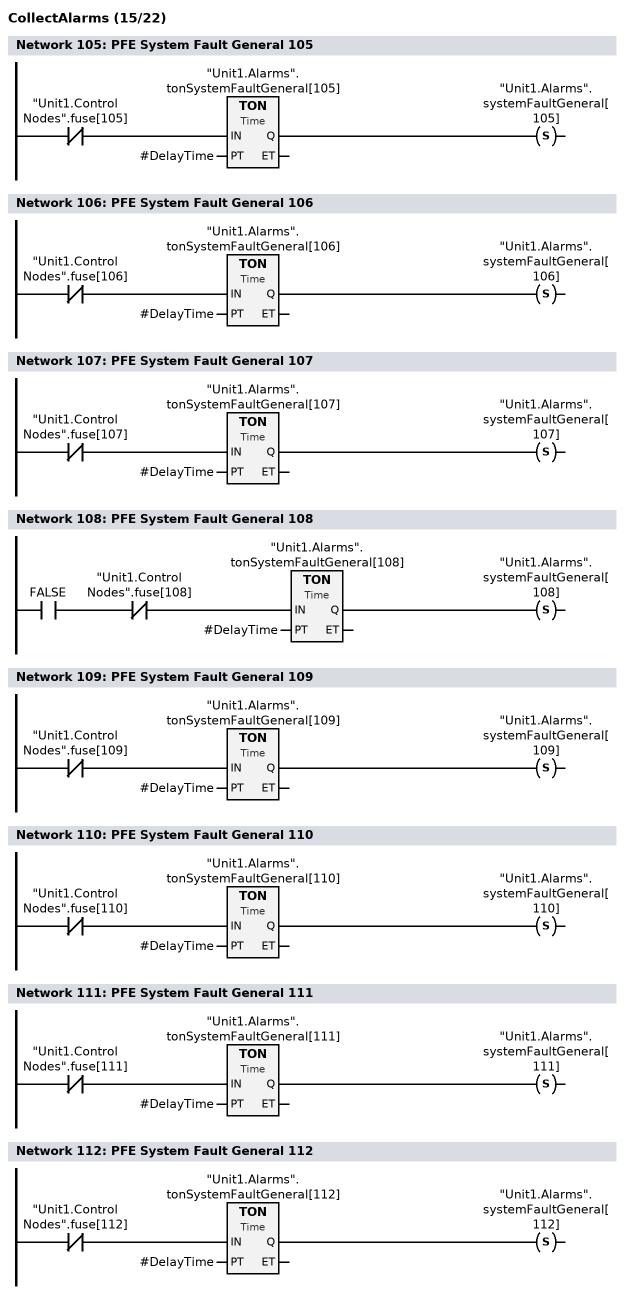
   RUNG wire#powerrail
      I_Contact( "Unit1.ControlNodes".fuse[105] )
      { S7_Templates := "time_type := Time" } "Unit1.Alarms".tonSystemFaultGeneral[105].TON(pt := #DelayTime, et =>)
      S_Coil( "Unit1.Alarms".systemFaultGeneral[105] )
   END_RUNG
   // the same network as SCL:
   "Unit1.Alarms".tonSystemFaultGeneral[105].TON(IN := NOT "Unit1.ControlNodes".fuse[105], PT := #DelayTime);
   IF "Unit1.Alarms".tonSystemFaultGeneral[105].Q THEN
       "Unit1.Alarms".systemFaultGeneral[105] := TRUE;
   END_IF;
END_REGION

REGION Network 106: PFE System Fault General 106
   RUNG wire#powerrail
      I_Contact( "Unit1.ControlNodes".fuse[106] )
      { S7_Templates := "time_type := Time" } "Unit1.Alarms".tonSystemFaultGeneral[106].TON(pt := #DelayTime, et =>)
      S_Coil( "Unit1.Alarms".systemFaultGeneral[106] )
   END_RUNG
   // the same network as SCL:
   "Unit1.Alarms".tonSystemFaultGeneral[106].TON(IN := NOT "Unit1.ControlNodes".fuse[106], PT := #DelayTime);
   IF "Unit1.Alarms".tonSystemFaultGeneral[106].Q THEN
       "Unit1.Alarms".systemFaultGeneral[106] := TRUE;
   END_IF;
END_REGION

REGION Network 107: PFE System Fault General 107
   RUNG wire#powerrail
      I_Contact( "Unit1.ControlNodes".fuse[107] )
      { S7_Templates := "time_type := Time" } "Unit1.Alarms".tonSystemFaultGeneral[107].TON(pt := #DelayTime, et =>)
      S_Coil( "Unit1.Alarms".systemFaultGeneral[107] )
   END_RUNG
   // the same network as SCL:
   "Unit1.Alarms".tonSystemFaultGeneral[107].TON(IN := NOT "Unit1.ControlNodes".fuse[107], PT := #DelayTime);
   IF "Unit1.Alarms".tonSystemFaultGeneral[107].Q THEN
       "Unit1.Alarms".systemFaultGeneral[107] := TRUE;
   END_IF;
END_REGION

REGION Network 108: PFE System Fault General 108
   RUNG wire#powerrail
      Contact( FALSE )
      I_Contact( "Unit1.ControlNodes".fuse[108] )
      { S7_Templates := "time_type := Time" } "Unit1.Alarms".tonSystemFaultGeneral[108].TON(pt := #DelayTime, et =>)
      S_Coil( "Unit1.Alarms".systemFaultGeneral[108] )
   END_RUNG
   // the same network as SCL:
   "Unit1.Alarms".tonSystemFaultGeneral[108].TON(IN := FALSE AND NOT "Unit1.ControlNodes".fuse[108],
                           PT := #DelayTime);
   IF "Unit1.Alarms".tonSystemFaultGeneral[108].Q THEN
       "Unit1.Alarms".systemFaultGeneral[108] := TRUE;
   END_IF;
END_REGION

REGION Network 109: PFE System Fault General 109
   RUNG wire#powerrail
      I_Contact( "Unit1.ControlNodes".fuse[109] )
      { S7_Templates := "time_type := Time" } "Unit1.Alarms".tonSystemFaultGeneral[109].TON(pt := #DelayTime, et =>)
      S_Coil( "Unit1.Alarms".systemFaultGeneral[109] )
   END_RUNG
   // the same network as SCL:
   "Unit1.Alarms".tonSystemFaultGeneral[109].TON(IN := NOT "Unit1.ControlNodes".fuse[109], PT := #DelayTime);
   IF "Unit1.Alarms".tonSystemFaultGeneral[109].Q THEN
       "Unit1.Alarms".systemFaultGeneral[109] := TRUE;
   END_IF;
END_REGION

REGION Network 110: PFE System Fault General 110
   RUNG wire#powerrail
      I_Contact( "Unit1.ControlNodes".fuse[110] )
      { S7_Templates := "time_type := Time" } "Unit1.Alarms".tonSystemFaultGeneral[110].TON(pt := #DelayTime, et =>)
      S_Coil( "Unit1.Alarms".systemFaultGeneral[110] )
   END_RUNG
   // the same network as SCL:
   "Unit1.Alarms".tonSystemFaultGeneral[110].TON(IN := NOT "Unit1.ControlNodes".fuse[110], PT := #DelayTime);
   IF "Unit1.Alarms".tonSystemFaultGeneral[110].Q THEN
       "Unit1.Alarms".systemFaultGeneral[110] := TRUE;
   END_IF;
END_REGION

REGION Network 111: PFE System Fault General 111
   RUNG wire#powerrail
      I_Contact( "Unit1.ControlNodes".fuse[111] )
      { S7_Templates := "time_type := Time" } "Unit1.Alarms".tonSystemFaultGeneral[111].TON(pt := #DelayTime, et =>)
      S_Coil( "Unit1.Alarms".systemFaultGeneral[111] )
   END_RUNG
   // the same network as SCL:
   "Unit1.Alarms".tonSystemFaultGeneral[111].TON(IN := NOT "Unit1.ControlNodes".fuse[111], PT := #DelayTime);
   IF "Unit1.Alarms".tonSystemFaultGeneral[111].Q THEN
       "Unit1.Alarms".systemFaultGeneral[111] := TRUE;
   END_IF;
END_REGION

REGION Network 112: PFE System Fault General 112
   RUNG wire#powerrail
      I_Contact( "Unit1.ControlNodes".fuse[112] )
      { S7_Templates := "time_type := Time" } "Unit1.Alarms".tonSystemFaultGeneral[112].TON(pt := #DelayTime, et =>)
      S_Coil( "Unit1.Alarms".systemFaultGeneral[112] )
   END_RUNG
   // the same network as SCL:
   "Unit1.Alarms".tonSystemFaultGeneral[112].TON(IN := NOT "Unit1.ControlNodes".fuse[112], PT := #DelayTime);
   IF "Unit1.Alarms".tonSystemFaultGeneral[112].Q THEN
       "Unit1.Alarms".systemFaultGeneral[112] := TRUE;
   END_IF;
END_REGION

REGION Network 113: PFE System Fault General 113
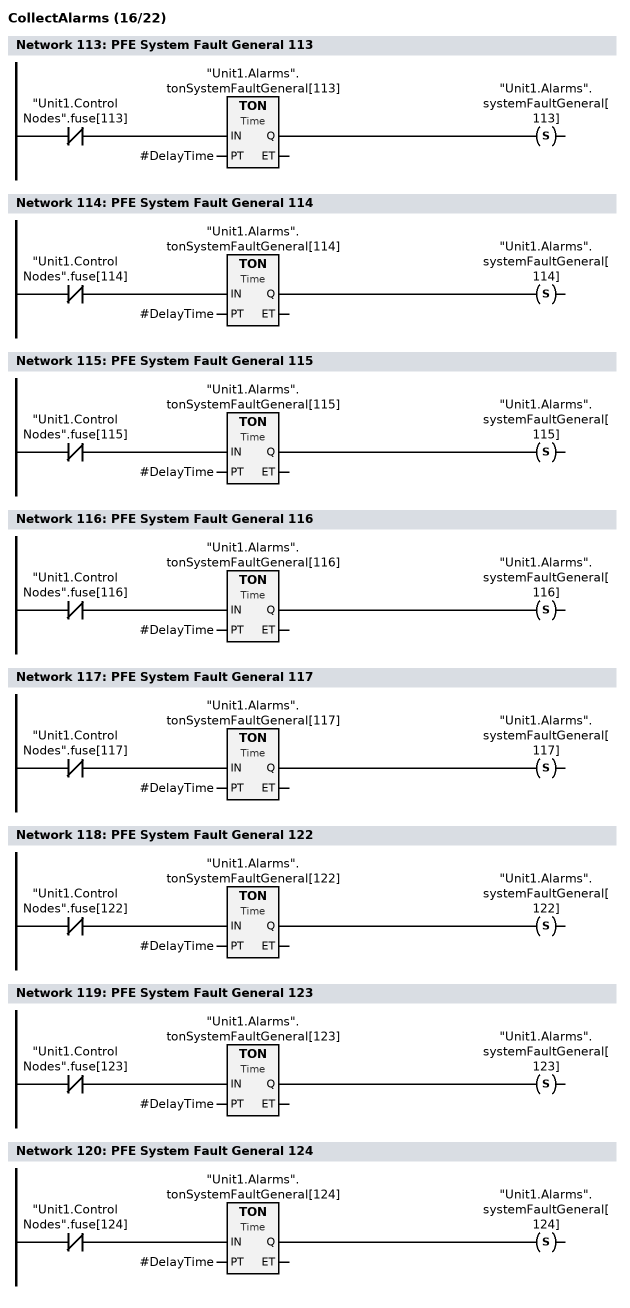
   RUNG wire#powerrail
      I_Contact( "Unit1.ControlNodes".fuse[113] )
      { S7_Templates := "time_type := Time" } "Unit1.Alarms".tonSystemFaultGeneral[113].TON(pt := #DelayTime, et =>)
      S_Coil( "Unit1.Alarms".systemFaultGeneral[113] )
   END_RUNG
   // the same network as SCL:
   "Unit1.Alarms".tonSystemFaultGeneral[113].TON(IN := NOT "Unit1.ControlNodes".fuse[113], PT := #DelayTime);
   IF "Unit1.Alarms".tonSystemFaultGeneral[113].Q THEN
       "Unit1.Alarms".systemFaultGeneral[113] := TRUE;
   END_IF;
END_REGION

REGION Network 114: PFE System Fault General 114
   RUNG wire#powerrail
      I_Contact( "Unit1.ControlNodes".fuse[114] )
      { S7_Templates := "time_type := Time" } "Unit1.Alarms".tonSystemFaultGeneral[114].TON(pt := #DelayTime, et =>)
      S_Coil( "Unit1.Alarms".systemFaultGeneral[114] )
   END_RUNG
   // the same network as SCL:
   "Unit1.Alarms".tonSystemFaultGeneral[114].TON(IN := NOT "Unit1.ControlNodes".fuse[114], PT := #DelayTime);
   IF "Unit1.Alarms".tonSystemFaultGeneral[114].Q THEN
       "Unit1.Alarms".systemFaultGeneral[114] := TRUE;
   END_IF;
END_REGION

REGION Network 115: PFE System Fault General 115
   RUNG wire#powerrail
      I_Contact( "Unit1.ControlNodes".fuse[115] )
      { S7_Templates := "time_type := Time" } "Unit1.Alarms".tonSystemFaultGeneral[115].TON(pt := #DelayTime, et =>)
      S_Coil( "Unit1.Alarms".systemFaultGeneral[115] )
   END_RUNG
   // the same network as SCL:
   "Unit1.Alarms".tonSystemFaultGeneral[115].TON(IN := NOT "Unit1.ControlNodes".fuse[115], PT := #DelayTime);
   IF "Unit1.Alarms".tonSystemFaultGeneral[115].Q THEN
       "Unit1.Alarms".systemFaultGeneral[115] := TRUE;
   END_IF;
END_REGION

REGION Network 116: PFE System Fault General 116
   RUNG wire#powerrail
      I_Contact( "Unit1.ControlNodes".fuse[116] )
      { S7_Templates := "time_type := Time" } "Unit1.Alarms".tonSystemFaultGeneral[116].TON(pt := #DelayTime, et =>)
      S_Coil( "Unit1.Alarms".systemFaultGeneral[116] )
   END_RUNG
   // the same network as SCL:
   "Unit1.Alarms".tonSystemFaultGeneral[116].TON(IN := NOT "Unit1.ControlNodes".fuse[116], PT := #DelayTime);
   IF "Unit1.Alarms".tonSystemFaultGeneral[116].Q THEN
       "Unit1.Alarms".systemFaultGeneral[116] := TRUE;
   END_IF;
END_REGION

REGION Network 117: PFE System Fault General 117
   RUNG wire#powerrail
      I_Contact( "Unit1.ControlNodes".fuse[117] )
      { S7_Templates := "time_type := Time" } "Unit1.Alarms".tonSystemFaultGeneral[117].TON(pt := #DelayTime, et =>)
      S_Coil( "Unit1.Alarms".systemFaultGeneral[117] )
   END_RUNG
   // the same network as SCL:
   "Unit1.Alarms".tonSystemFaultGeneral[117].TON(IN := NOT "Unit1.ControlNodes".fuse[117], PT := #DelayTime);
   IF "Unit1.Alarms".tonSystemFaultGeneral[117].Q THEN
       "Unit1.Alarms".systemFaultGeneral[117] := TRUE;
   END_IF;
END_REGION

REGION Network 118: PFE System Fault General 122
   RUNG wire#powerrail
      I_Contact( "Unit1.ControlNodes".fuse[122] )
      { S7_Templates := "time_type := Time" } "Unit1.Alarms".tonSystemFaultGeneral[122].TON(pt := #DelayTime, et =>)
      S_Coil( "Unit1.Alarms".systemFaultGeneral[122] )
   END_RUNG
   // the same network as SCL:
   "Unit1.Alarms".tonSystemFaultGeneral[122].TON(IN := NOT "Unit1.ControlNodes".fuse[122], PT := #DelayTime);
   IF "Unit1.Alarms".tonSystemFaultGeneral[122].Q THEN
       "Unit1.Alarms".systemFaultGeneral[122] := TRUE;
   END_IF;
END_REGION

REGION Network 119: PFE System Fault General 123
   RUNG wire#powerrail
      I_Contact( "Unit1.ControlNodes".fuse[123] )
      { S7_Templates := "time_type := Time" } "Unit1.Alarms".tonSystemFaultGeneral[123].TON(pt := #DelayTime, et =>)
      S_Coil( "Unit1.Alarms".systemFaultGeneral[123] )
   END_RUNG
   // the same network as SCL:
   "Unit1.Alarms".tonSystemFaultGeneral[123].TON(IN := NOT "Unit1.ControlNodes".fuse[123], PT := #DelayTime);
   IF "Unit1.Alarms".tonSystemFaultGeneral[123].Q THEN
       "Unit1.Alarms".systemFaultGeneral[123] := TRUE;
   END_IF;
END_REGION

REGION Network 120: PFE System Fault General 124
   RUNG wire#powerrail
      I_Contact( "Unit1.ControlNodes".fuse[124] )
      { S7_Templates := "time_type := Time" } "Unit1.Alarms".tonSystemFaultGeneral[124].TON(pt := #DelayTime, et =>)
      S_Coil( "Unit1.Alarms".systemFaultGeneral[124] )
   END_RUNG
   // the same network as SCL:
   "Unit1.Alarms".tonSystemFaultGeneral[124].TON(IN := NOT "Unit1.ControlNodes".fuse[124], PT := #DelayTime);
   IF "Unit1.Alarms".tonSystemFaultGeneral[124].Q THEN
       "Unit1.Alarms".systemFaultGeneral[124] := TRUE;
   END_IF;
END_REGION

REGION Network 121: PFE System Fault General 125
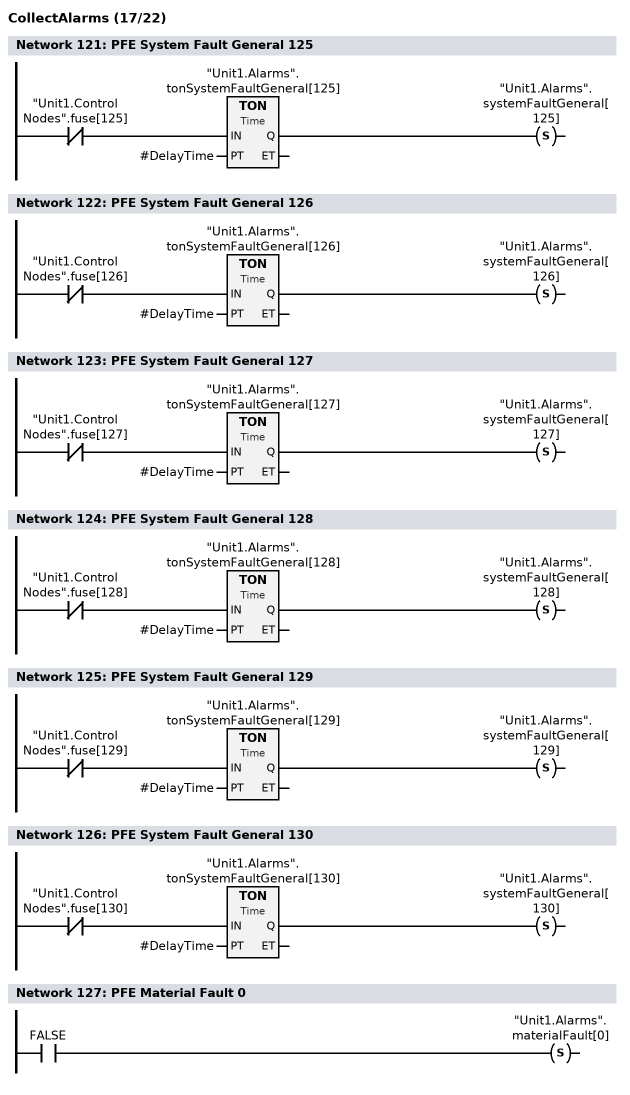
   RUNG wire#powerrail
      I_Contact( "Unit1.ControlNodes".fuse[125] )
      { S7_Templates := "time_type := Time" } "Unit1.Alarms".tonSystemFaultGeneral[125].TON(pt := #DelayTime, et =>)
      S_Coil( "Unit1.Alarms".systemFaultGeneral[125] )
   END_RUNG
   // the same network as SCL:
   "Unit1.Alarms".tonSystemFaultGeneral[125].TON(IN := NOT "Unit1.ControlNodes".fuse[125], PT := #DelayTime);
   IF "Unit1.Alarms".tonSystemFaultGeneral[125].Q THEN
       "Unit1.Alarms".systemFaultGeneral[125] := TRUE;
   END_IF;
END_REGION

REGION Network 122: PFE System Fault General 126
   RUNG wire#powerrail
      I_Contact( "Unit1.ControlNodes".fuse[126] )
      { S7_Templates := "time_type := Time" } "Unit1.Alarms".tonSystemFaultGeneral[126].TON(pt := #DelayTime, et =>)
      S_Coil( "Unit1.Alarms".systemFaultGeneral[126] )
   END_RUNG
   // the same network as SCL:
   "Unit1.Alarms".tonSystemFaultGeneral[126].TON(IN := NOT "Unit1.ControlNodes".fuse[126], PT := #DelayTime);
   IF "Unit1.Alarms".tonSystemFaultGeneral[126].Q THEN
       "Unit1.Alarms".systemFaultGeneral[126] := TRUE;
   END_IF;
END_REGION

REGION Network 123: PFE System Fault General 127
   RUNG wire#powerrail
      I_Contact( "Unit1.ControlNodes".fuse[127] )
      { S7_Templates := "time_type := Time" } "Unit1.Alarms".tonSystemFaultGeneral[127].TON(pt := #DelayTime, et =>)
      S_Coil( "Unit1.Alarms".systemFaultGeneral[127] )
   END_RUNG
   // the same network as SCL:
   "Unit1.Alarms".tonSystemFaultGeneral[127].TON(IN := NOT "Unit1.ControlNodes".fuse[127], PT := #DelayTime);
   IF "Unit1.Alarms".tonSystemFaultGeneral[127].Q THEN
       "Unit1.Alarms".systemFaultGeneral[127] := TRUE;
   END_IF;
END_REGION

REGION Network 124: PFE System Fault General 128
   RUNG wire#powerrail
      I_Contact( "Unit1.ControlNodes".fuse[128] )
      { S7_Templates := "time_type := Time" } "Unit1.Alarms".tonSystemFaultGeneral[128].TON(pt := #DelayTime, et =>)
      S_Coil( "Unit1.Alarms".systemFaultGeneral[128] )
   END_RUNG
   // the same network as SCL:
   "Unit1.Alarms".tonSystemFaultGeneral[128].TON(IN := NOT "Unit1.ControlNodes".fuse[128], PT := #DelayTime);
   IF "Unit1.Alarms".tonSystemFaultGeneral[128].Q THEN
       "Unit1.Alarms".systemFaultGeneral[128] := TRUE;
   END_IF;
END_REGION

REGION Network 125: PFE System Fault General 129
   RUNG wire#powerrail
      I_Contact( "Unit1.ControlNodes".fuse[129] )
      { S7_Templates := "time_type := Time" } "Unit1.Alarms".tonSystemFaultGeneral[129].TON(pt := #DelayTime, et =>)
      S_Coil( "Unit1.Alarms".systemFaultGeneral[129] )
   END_RUNG
   // the same network as SCL:
   "Unit1.Alarms".tonSystemFaultGeneral[129].TON(IN := NOT "Unit1.ControlNodes".fuse[129], PT := #DelayTime);
   IF "Unit1.Alarms".tonSystemFaultGeneral[129].Q THEN
       "Unit1.Alarms".systemFaultGeneral[129] := TRUE;
   END_IF;
END_REGION

REGION Network 126: PFE System Fault General 130
   RUNG wire#powerrail
      I_Contact( "Unit1.ControlNodes".fuse[130] )
      { S7_Templates := "time_type := Time" } "Unit1.Alarms".tonSystemFaultGeneral[130].TON(pt := #DelayTime, et =>)
      S_Coil( "Unit1.Alarms".systemFaultGeneral[130] )
   END_RUNG
   // the same network as SCL:
   "Unit1.Alarms".tonSystemFaultGeneral[130].TON(IN := NOT "Unit1.ControlNodes".fuse[130], PT := #DelayTime);
   IF "Unit1.Alarms".tonSystemFaultGeneral[130].Q THEN
       "Unit1.Alarms".systemFaultGeneral[130] := TRUE;
   END_IF;
END_REGION

REGION Network 127: PFE Material Fault 0
   RUNG wire#powerrail
      Contact( FALSE )
      S_Coil( "Unit1.Alarms".materialFault[0] )
   END_RUNG
   // the same network as SCL:
   IF FALSE THEN "Unit1.Alarms".materialFault[0] := TRUE; END_IF;
END_REGION

REGION Network 129: *************** Warning **************************
END_REGION

REGION Network 130: PFE Maintenance Warnings
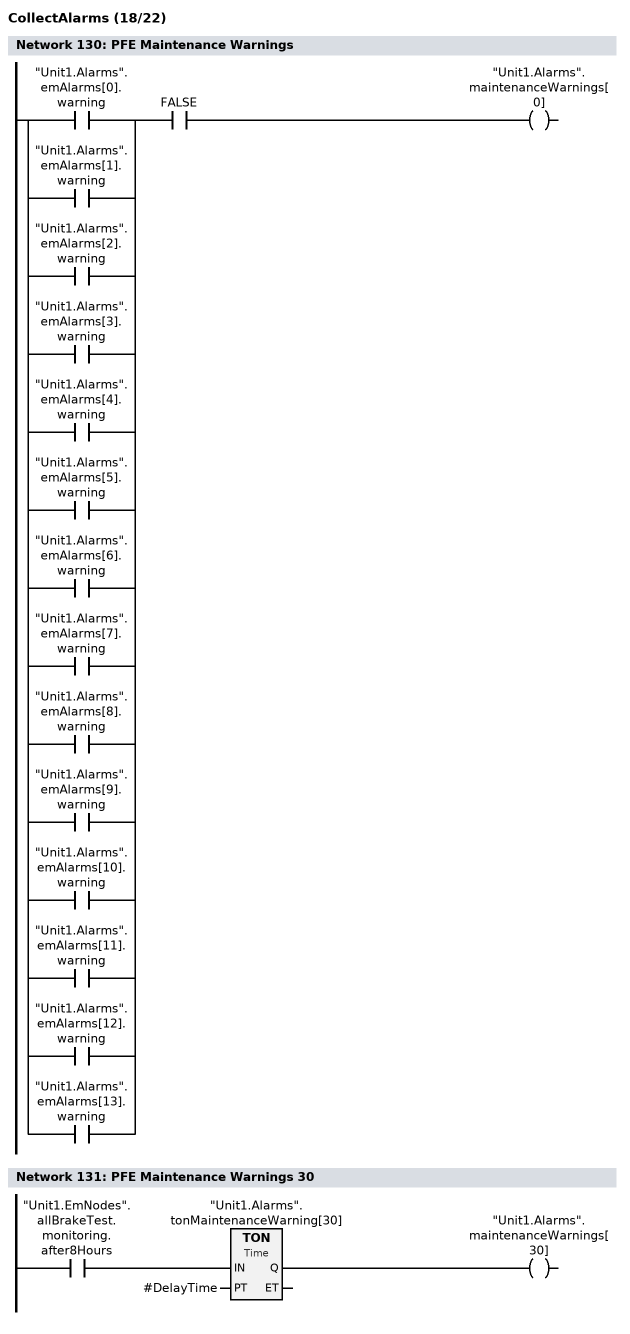
   RUNG wire#powerrail
      Contact( "Unit1.Alarms".emAlarms[0].warning )
      wire#w1
      Contact( FALSE )
      Coil( "Unit1.Alarms".maintenanceWarnings[0] )
   END_RUNG
   RUNG wire#powerrail
      Contact( "Unit1.Alarms".emAlarms[1].warning )
   END_RUNG wire#w1
   RUNG wire#powerrail
      Contact( "Unit1.Alarms".emAlarms[2].warning )
   END_RUNG wire#w1
   RUNG wire#powerrail
      Contact( "Unit1.Alarms".emAlarms[3].warning )
   END_RUNG wire#w1
   RUNG wire#powerrail
      Contact( "Unit1.Alarms".emAlarms[4].warning )
   END_RUNG wire#w1
   RUNG wire#powerrail
      Contact( "Unit1.Alarms".emAlarms[5].warning )
   END_RUNG wire#w1
   RUNG wire#powerrail
      Contact( "Unit1.Alarms".emAlarms[6].warning )
   END_RUNG wire#w1
   RUNG wire#powerrail
      Contact( "Unit1.Alarms".emAlarms[7].warning )
   END_RUNG wire#w1
   RUNG wire#powerrail
      Contact( "Unit1.Alarms".emAlarms[8].warning )
   END_RUNG wire#w1
   RUNG wire#powerrail
      Contact( "Unit1.Alarms".emAlarms[9].warning )
   END_RUNG wire#w1
   RUNG wire#powerrail
      Contact( "Unit1.Alarms".emAlarms[10].warning )
   END_RUNG wire#w1
   RUNG wire#powerrail
      Contact( "Unit1.Alarms".emAlarms[11].warning )
   END_RUNG wire#w1
   RUNG wire#powerrail
      Contact( "Unit1.Alarms".emAlarms[12].warning )
   END_RUNG wire#w1
   RUNG wire#powerrail
      Contact( "Unit1.Alarms".emAlarms[13].warning )
   END_RUNG wire#w1
   // the same network as SCL:
   "Unit1.Alarms".maintenanceWarnings[0] := ("Unit1.Alarms".emAlarms[0].warning OR "Unit1.Alarms".emAlarms[1].warning OR "Unit1.Alarms".emAlarms[2].warning OR "Unit1.Alarms".emAlarms[3].warning OR "Unit1.Alarms".emAlarms[4].warning OR "Unit1.Alarms".emAlarms[5].warning OR "Unit1.Alarms".emAlarms[6].warning OR "Unit1.Alarms".emAlarms[7].warning OR "Unit1.Alarms".emAlarms[8].warning OR "Unit1.Alarms".emAlarms[9].warning OR "Unit1.Alarms".emAlarms[10].warning OR "Unit1.Alarms".emAlarms[11].warning OR "Unit1.Alarms".emAlarms[12].warning OR "Unit1.Alarms".emAlarms[13].warning) AND FALSE;
END_REGION

REGION Network 131: PFE Maintenance Warnings 30
   RUNG wire#powerrail
      Contact( "Unit1.EmNodes".allBrakeTest.monitoring.after8Hours )
      { S7_Templates := "time_type := Time" } "Unit1.Alarms".tonMaintenanceWarning[30].TON(pt := #DelayTime, et =>)
      Coil( "Unit1.Alarms".maintenanceWarnings[30] )
   END_RUNG
   // the same network as SCL:
   "Unit1.Alarms".tonMaintenanceWarning[30].TON(IN := "Unit1.EmNodes".allBrakeTest.monitoring.after8Hours,
                           PT := #DelayTime);
   "Unit1.Alarms".maintenanceWarnings[30] := "Unit1.Alarms".tonMaintenanceWarning[30].Q;
END_REGION

REGION Network 132: PFE Maintenance Warnings 31
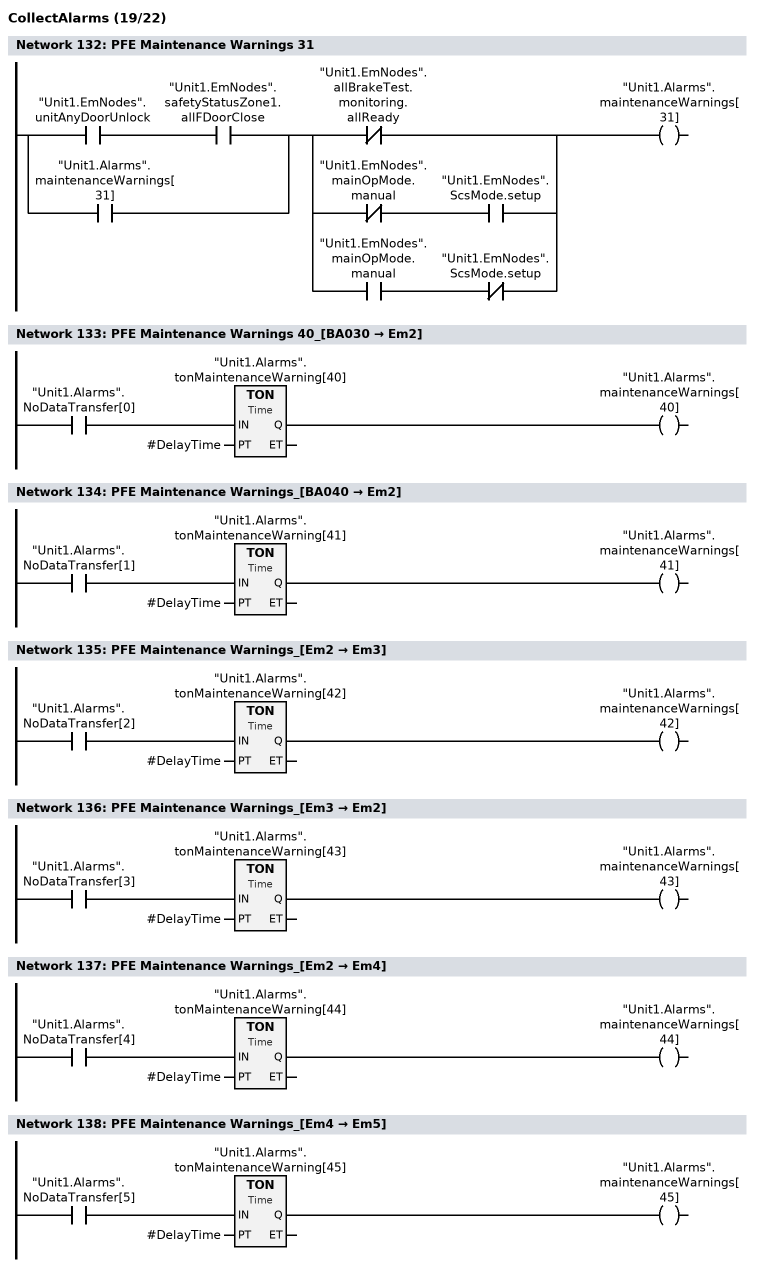
   RUNG wire#powerrail
      Contact( "Unit1.EmNodes".unitAnyDoorUnlock )
      Contact( "Unit1.EmNodes".safetyStatusZone1.allFDoorClose )
      wire#w1
      I_Contact( "Unit1.EmNodes".allBrakeTest.monitoring.allReady )
      wire#w2
      Coil( "Unit1.Alarms".maintenanceWarnings[31] )
   END_RUNG
   RUNG wire#powerrail
      Contact( "Unit1.Alarms".maintenanceWarnings[31] )
   END_RUNG wire#w1
   RUNG wire#w1
      I_Contact( "Unit1.EmNodes".mainOpMode.manual )
      Contact( "Unit1.EmNodes".ScsMode.setup )
   END_RUNG wire#w2
   RUNG wire#w1
      Contact( "Unit1.EmNodes".mainOpMode.manual )
      I_Contact( "Unit1.EmNodes".ScsMode.setup )
   END_RUNG wire#w2
   // the same network as SCL:
   "Unit1.Alarms".maintenanceWarnings[31] := (("Unit1.EmNodes".unitAnyDoorUnlock AND "Unit1.EmNodes".safetyStatusZone1.allFDoorClose) OR "Unit1.Alarms".maintenanceWarnings[31]) AND (NOT "Unit1.EmNodes".allBrakeTest.monitoring.allReady OR (NOT "Unit1.EmNodes".mainOpMode.manual AND "Unit1.EmNodes".ScsMode.setup) OR ("Unit1.EmNodes".mainOpMode.manual AND NOT "Unit1.EmNodes".ScsMode.setup));
END_REGION

REGION Network 133: PFE Maintenance Warnings 40_[BA030 → Em2]
   RUNG wire#powerrail
      Contact( "Unit1.Alarms".NoDataTransfer[0] )
      { S7_Templates := "time_type := Time" } "Unit1.Alarms".tonMaintenanceWarning[40].TON(pt := #DelayTime, et =>)
      Coil( "Unit1.Alarms".maintenanceWarnings[40] )
   END_RUNG
   // the same network as SCL:
   "Unit1.Alarms".tonMaintenanceWarning[40].TON(IN := "Unit1.Alarms".NoDataTransfer[0], PT := #DelayTime);
   "Unit1.Alarms".maintenanceWarnings[40] := "Unit1.Alarms".tonMaintenanceWarning[40].Q;
END_REGION

REGION Network 134: PFE Maintenance Warnings_[BA040 → Em2]
   RUNG wire#powerrail
      Contact( "Unit1.Alarms".NoDataTransfer[1] )
      { S7_Templates := "time_type := Time" } "Unit1.Alarms".tonMaintenanceWarning[41].TON(pt := #DelayTime, et =>)
      Coil( "Unit1.Alarms".maintenanceWarnings[41] )
   END_RUNG
   // the same network as SCL:
   "Unit1.Alarms".tonMaintenanceWarning[41].TON(IN := "Unit1.Alarms".NoDataTransfer[1], PT := #DelayTime);
   "Unit1.Alarms".maintenanceWarnings[41] := "Unit1.Alarms".tonMaintenanceWarning[41].Q;
END_REGION

REGION Network 135: PFE Maintenance Warnings_[Em2 → Em3]
   RUNG wire#powerrail
      Contact( "Unit1.Alarms".NoDataTransfer[2] )
      { S7_Templates := "time_type := Time" } "Unit1.Alarms".tonMaintenanceWarning[42].TON(pt := #DelayTime, et =>)
      Coil( "Unit1.Alarms".maintenanceWarnings[42] )
   END_RUNG
   // the same network as SCL:
   "Unit1.Alarms".tonMaintenanceWarning[42].TON(IN := "Unit1.Alarms".NoDataTransfer[2], PT := #DelayTime);
   "Unit1.Alarms".maintenanceWarnings[42] := "Unit1.Alarms".tonMaintenanceWarning[42].Q;
END_REGION

REGION Network 136: PFE Maintenance Warnings_[Em3 → Em2]
   RUNG wire#powerrail
      Contact( "Unit1.Alarms".NoDataTransfer[3] )
      { S7_Templates := "time_type := Time" } "Unit1.Alarms".tonMaintenanceWarning[43].TON(pt := #DelayTime, et =>)
      Coil( "Unit1.Alarms".maintenanceWarnings[43] )
   END_RUNG
   // the same network as SCL:
   "Unit1.Alarms".tonMaintenanceWarning[43].TON(IN := "Unit1.Alarms".NoDataTransfer[3], PT := #DelayTime);
   "Unit1.Alarms".maintenanceWarnings[43] := "Unit1.Alarms".tonMaintenanceWarning[43].Q;
END_REGION

REGION Network 137: PFE Maintenance Warnings_[Em2 → Em4]
   RUNG wire#powerrail
      Contact( "Unit1.Alarms".NoDataTransfer[4] )
      { S7_Templates := "time_type := Time" } "Unit1.Alarms".tonMaintenanceWarning[44].TON(pt := #DelayTime, et =>)
      Coil( "Unit1.Alarms".maintenanceWarnings[44] )
   END_RUNG
   // the same network as SCL:
   "Unit1.Alarms".tonMaintenanceWarning[44].TON(IN := "Unit1.Alarms".NoDataTransfer[4], PT := #DelayTime);
   "Unit1.Alarms".maintenanceWarnings[44] := "Unit1.Alarms".tonMaintenanceWarning[44].Q;
END_REGION

REGION Network 138: PFE Maintenance Warnings_[Em4 → Em5]
   RUNG wire#powerrail
      Contact( "Unit1.Alarms".NoDataTransfer[5] )
      { S7_Templates := "time_type := Time" } "Unit1.Alarms".tonMaintenanceWarning[45].TON(pt := #DelayTime, et =>)
      Coil( "Unit1.Alarms".maintenanceWarnings[45] )
   END_RUNG
   // the same network as SCL:
   "Unit1.Alarms".tonMaintenanceWarning[45].TON(IN := "Unit1.Alarms".NoDataTransfer[5], PT := #DelayTime);
   "Unit1.Alarms".maintenanceWarnings[45] := "Unit1.Alarms".tonMaintenanceWarning[45].Q;
END_REGION

REGION Network 139: PFE Maintenance Warnings_[Em5 → Em6]
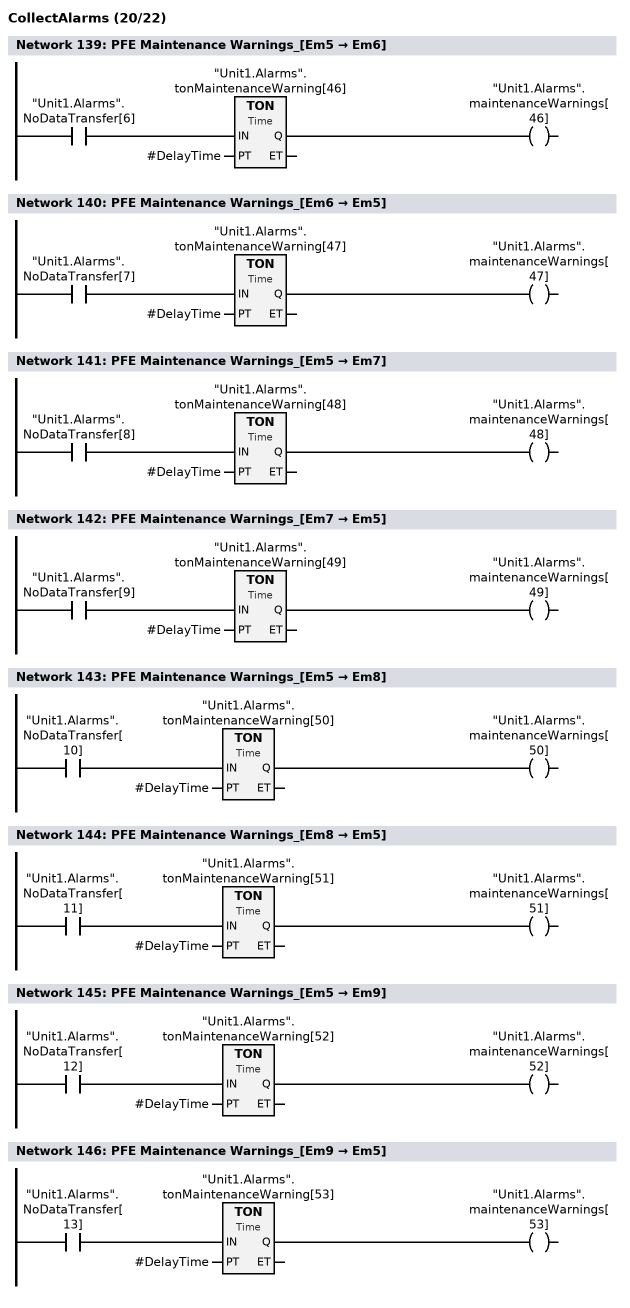
   RUNG wire#powerrail
      Contact( "Unit1.Alarms".NoDataTransfer[6] )
      { S7_Templates := "time_type := Time" } "Unit1.Alarms".tonMaintenanceWarning[46].TON(pt := #DelayTime, et =>)
      Coil( "Unit1.Alarms".maintenanceWarnings[46] )
   END_RUNG
   // the same network as SCL:
   "Unit1.Alarms".tonMaintenanceWarning[46].TON(IN := "Unit1.Alarms".NoDataTransfer[6], PT := #DelayTime);
   "Unit1.Alarms".maintenanceWarnings[46] := "Unit1.Alarms".tonMaintenanceWarning[46].Q;
END_REGION

REGION Network 140: PFE Maintenance Warnings_[Em6 → Em5]
   RUNG wire#powerrail
      Contact( "Unit1.Alarms".NoDataTransfer[7] )
      { S7_Templates := "time_type := Time" } "Unit1.Alarms".tonMaintenanceWarning[47].TON(pt := #DelayTime, et =>)
      Coil( "Unit1.Alarms".maintenanceWarnings[47] )
   END_RUNG
   // the same network as SCL:
   "Unit1.Alarms".tonMaintenanceWarning[47].TON(IN := "Unit1.Alarms".NoDataTransfer[7], PT := #DelayTime);
   "Unit1.Alarms".maintenanceWarnings[47] := "Unit1.Alarms".tonMaintenanceWarning[47].Q;
END_REGION

REGION Network 141: PFE Maintenance Warnings_[Em5 → Em7]
   RUNG wire#powerrail
      Contact( "Unit1.Alarms".NoDataTransfer[8] )
      { S7_Templates := "time_type := Time" } "Unit1.Alarms".tonMaintenanceWarning[48].TON(pt := #DelayTime, et =>)
      Coil( "Unit1.Alarms".maintenanceWarnings[48] )
   END_RUNG
   // the same network as SCL:
   "Unit1.Alarms".tonMaintenanceWarning[48].TON(IN := "Unit1.Alarms".NoDataTransfer[8], PT := #DelayTime);
   "Unit1.Alarms".maintenanceWarnings[48] := "Unit1.Alarms".tonMaintenanceWarning[48].Q;
END_REGION

REGION Network 142: PFE Maintenance Warnings_[Em7 → Em5]
   RUNG wire#powerrail
      Contact( "Unit1.Alarms".NoDataTransfer[9] )
      { S7_Templates := "time_type := Time" } "Unit1.Alarms".tonMaintenanceWarning[49].TON(pt := #DelayTime, et =>)
      Coil( "Unit1.Alarms".maintenanceWarnings[49] )
   END_RUNG
   // the same network as SCL:
   "Unit1.Alarms".tonMaintenanceWarning[49].TON(IN := "Unit1.Alarms".NoDataTransfer[9], PT := #DelayTime);
   "Unit1.Alarms".maintenanceWarnings[49] := "Unit1.Alarms".tonMaintenanceWarning[49].Q;
END_REGION

REGION Network 143: PFE Maintenance Warnings_[Em5 → Em8]
   RUNG wire#powerrail
      Contact( "Unit1.Alarms".NoDataTransfer[10] )
      { S7_Templates := "time_type := Time" } "Unit1.Alarms".tonMaintenanceWarning[50].TON(pt := #DelayTime, et =>)
      Coil( "Unit1.Alarms".maintenanceWarnings[50] )
   END_RUNG
   // the same network as SCL:
   "Unit1.Alarms".tonMaintenanceWarning[50].TON(IN := "Unit1.Alarms".NoDataTransfer[10], PT := #DelayTime);
   "Unit1.Alarms".maintenanceWarnings[50] := "Unit1.Alarms".tonMaintenanceWarning[50].Q;
END_REGION

REGION Network 144: PFE Maintenance Warnings_[Em8 → Em5]
   RUNG wire#powerrail
      Contact( "Unit1.Alarms".NoDataTransfer[11] )
      { S7_Templates := "time_type := Time" } "Unit1.Alarms".tonMaintenanceWarning[51].TON(pt := #DelayTime, et =>)
      Coil( "Unit1.Alarms".maintenanceWarnings[51] )
   END_RUNG
   // the same network as SCL:
   "Unit1.Alarms".tonMaintenanceWarning[51].TON(IN := "Unit1.Alarms".NoDataTransfer[11], PT := #DelayTime);
   "Unit1.Alarms".maintenanceWarnings[51] := "Unit1.Alarms".tonMaintenanceWarning[51].Q;
END_REGION

